// TwinCAT 3 PLC project plc_kfe_gatt
// ProgramVersion: 3.1.4023.0
// libraries:
//   L2SI Vacuum Library, * (SLAC)
//   LCLS General, * (SLAC)
//   lcls-twincat-motion, * (SLAC)
//   PMPS, * (SLAC - LCLS)
//   Tc2_ControllerToolbox, * (Beckhoff Automation GmbH)
//   Tc2_EtherCAT, * (Beckhoff Automation GmbH)
//   Tc2_MC2, * (Beckhoff Automation GmbH)
//   Tc2_Standard, * (Beckhoff Automation GmbH)
//   Tc2_System, * (Beckhoff Automation GmbH)
//   Tc2_Utilities, * (Beckhoff Automation GmbH)
//   Tc3_Module, * (Beckhoff Automation GmbH)
// project tree:
//   DUTs/ E_HomeState.TcDUT, E_MoveState.TcDUT, ST_VGP.TcDUT
//   GVLs/ GVL_Devices.TcGVL, GVL_GATT.TcGVL, GVL_ILK.TcGVL, GVL_MOT.TcGVL, GVL_Variables.TcGVL, Main.TcGVL
//   / PlcTask.TcTTO
//   POUs/ DIAGNOSTICS.TcPOU, FB_MAA_States.TcPOU, FB_VGP.TcPOU, PRG_1_PlcTask.TcPOU, PRG_GATT.TcPOU, PRG_INJ.TcPOU, PRG_Motion.TcPOU, PRG_Motors_Test.TcPOU, PRG_VGP.TcPOU
// real-time tasks:
//   TASK PlcTask: cycle T#10ms, priority 20, ADS port 350
// motion (NC):
//   TASK NC-Task 1 SAF: cycle T#2ms, priority 4, ADS port 501
//   TASK NC-Task 1 SVB: cycle T#10ms, priority 8, ADS port 511
//   AXIS MA_1_X (id 1)
//     Velo: Maximum=5
//     OtherSettings: AllowMotionCmdToSlave=true
//     encoder EncType=4
//       EncPara: ScaleFactorNumerator=6.1991875e-05, MaxCount=#x0000ffff
//         Inc: RefSoftSyncMask=#x0000ffff
//     drive DrvType=24
//       Analog: VeloReferenz=7.93496, TorqueScale=10, ScaleFactorActTorque=0.1
//       TimeComp: TaskDelayCycles=1
//     controller CtrType=1
//       CtrPara: PriorControlFactor=1
//         Observer: BandWidth=20
//   AXIS MA_1_Y (id 2)
//     Dynamic: AccelerationMaximum=30, DecelerationMaximum=30
//     Velo: Maximum=40
//     OtherSettings: AllowMotionCmdToSlave=true
//     encoder EncType=4
//       EncPara: ScaleFactorNumerator=0.000390625, MaxCount=#x0000ffff
//         Inc: RefSoftSyncMask=#x0000ffff
//     drive DrvType=24
//       Analog: VeloReferenz=50, TorqueScale=10, ScaleFactorActTorque=0.1
//       TimeComp: TaskDelayCycles=1
//     controller CtrType=1
//       CtrPara: PriorControlFactor=1
//         Observer: BandWidth=20
//   AXIS MA_2_X (id 3)
//     Velo: Maximum=5
//     OtherSettings: AllowMotionCmdToSlave=true
//     encoder EncType=4
//       EncPara: ScaleFactorNumerator=6.1991875e-05, MaxCount=#x0000ffff
//         Inc: RefSoftSyncMask=#x0000ffff
//     drive DrvType=24
//       Analog: VeloReferenz=7.93496, TorqueScale=10, ScaleFactorActTorque=0.1
//       TimeComp: TaskDelayCycles=1
//     controller CtrType=1
//       CtrPara: PriorControlFactor=1
//         Observer: BandWidth=20
//   AXIS MA_2_Y (id 4)
//     Dynamic: AccelerationMaximum=30, DecelerationMaximum=30
//     Velo: Maximum=40
//     OtherSettings: AllowMotionCmdToSlave=true
//     encoder EncType=4
//       EncPara: ScaleFactorNumerator=0.000390625, MaxCount=#x0000ffff
//         Inc: RefSoftSyncMask=#x0000ffff
//     drive DrvType=24
//       Analog: VeloReferenz=50, TorqueScale=10, ScaleFactorActTorque=0.1
//       TimeComp: TaskDelayCycles=1
//     controller CtrType=1
//       CtrPara: PriorControlFactor=1
//         Observer: BandWidth=20
//   AXIS MA_3_X (id 5)
//     Velo: Maximum=5
//     OtherSettings: AllowMotionCmdToSlave=true
//     encoder EncType=4
//       EncPara: ScaleFactorNumerator=6.1991875e-05, MaxCount=#x0000ffff
//         Inc: RefSoftSyncMask=#x0000ffff
//     drive DrvType=24
//       Analog: VeloReferenz=7.93496, TorqueScale=10, ScaleFactorActTorque=0.1
//       TimeComp: TaskDelayCycles=1
//     controller CtrType=1
//       CtrPara: PriorControlFactor=1
//         Observer: BandWidth=20
//   AXIS MA_3_Y (id 6)
//     Dynamic: AccelerationMaximum=30, DecelerationMaximum=30
//     Velo: Maximum=40
//     OtherSettings: AllowMotionCmdToSlave=true
//     encoder EncType=4
//       EncPara: ScaleFactorNumerator=0.000390625, MaxCount=#x0000ffff
//         Inc: RefSoftSyncMask=#x0000ffff
//     drive DrvType=24
//       Analog: VeloReferenz=50, TorqueScale=10, ScaleFactorActTorque=0.1
//       TimeComp: TaskDelayCycles=1
//     controller CtrType=1
//       CtrPara: PriorControlFactor=1
//         Observer: BandWidth=20
//   AXIS MA_4_X (id 7)
//     Velo: Maximum=5
//     OtherSettings: AllowMotionCmdToSlave=true
//     encoder EncType=4
//       EncPara: ScaleFactorNumerator=6.1991875e-05, MaxCount=#x0000ffff
//         Inc: RefSoftSyncMask=#x0000ffff
//     drive DrvType=24
//       Analog: VeloReferenz=7.93496, TorqueScale=10, ScaleFactorActTorque=0.1
//       TimeComp: TaskDelayCycles=1
//     controller CtrType=1
//       CtrPara: PriorControlFactor=1
//         Observer: BandWidth=20
//   AXIS MA_4_Y (id 8)
//     Dynamic: AccelerationMaximum=30, DecelerationMaximum=30
//     Velo: Maximum=40
//     OtherSettings: AllowMotionCmdToSlave=true
//     encoder EncType=4
//       EncPara: ScaleFactorNumerator=0.000390625, MaxCount=#x0000ffff
//         Inc: RefSoftSyncMask=#x0000ffff
//     drive DrvType=24
//       Analog: VeloReferenz=50, TorqueScale=10, ScaleFactorActTorque=0.1
//       TimeComp: TaskDelayCycles=1
//     controller CtrType=1
//       CtrPara: PriorControlFactor=1
//         Observer: BandWidth=20
//   AXIS VGP_80 (id 9)
//     Velo: Maximum=1800
//     OtherSettings: AllowMotionCmdToSlave=true
//     encoder EncType=4
//       EncPara: ScaleFactorNumerator=0.0390625, Inverse=true, MaxCount=#x0000ffff
//         Inc: RefSoftSyncMask=#x0000ffff
//     drive DrvType=24
//       Analog: VeloReferenz=2000, TorqueScale=10, ScaleFactorActTorque=0.1
//       TimeComp: TaskDelayCycles=1
//     controller CtrType=1
//       CtrPara: PriorControlFactor=1
//         Observer: BandWidth=20
// I/O:
//   DEVICE =+-CX2020/EtherCAT1, AmsNetId 172.21.92.57.2.1
//     =+-EK1200_00_00 [EK1200-5000 EtherCAT Power supply (2A E-Bus)]
//       =+-ES3064_00_01 [EL3064 4Ch. Ana. Input 0-10V]
//       =+-ES9070_00_02 [EL9070 Shield terminal]
//       =+-ES1008_00_03 [EL1008 8Ch. Dig. Input 24V, 3ms]
//       =+-ES2008_00_05 [EL2008 8Ch. Dig. Output 24V, 0.5A]
//       =+-EL2794_00_06 [EL2794 4Ch. Dig. Output 24V AC/DC, 2A, short-circuit-proof]
//       =+-ES2202_00_07 [EL2202 2Ch. Dig. Output 24V, 0.5A]
//       =+-EL6692_00_08 [EL6692 EtherCAT Bridge terminal (Primary)]
//       =+-EK1110_00_09 [EK1110 EtherCAT extension]
//     =+-EK1100_01_00 [EK1100 EtherCAT Coupler (2A E-Bus)]
//       =+-ES3064_01_01 [EL3064 4Ch. Ana. Input 0-10V]
//       =+-ES3064_01_02 [EL3064 4Ch. Ana. Input 0-10V]
//       =+-EL2798_01_03 [EL2798 8Ch. Dig. Output 24V AC/DC, 2A, potential-free]
//       =+-ES3064_01_04 [EL3064 4Ch. Ana. Input 0-10V]
//       =+-ES3064_01_05 [EL3064 4Ch. Ana. Input 0-10V]
//       =+-ES3064_01_06 [EL3064 4Ch. Ana. Input 0-10V]
//       =+-ES3064_01_07 [EL3064 4Ch. Ana. Input 0-10V]
//       =+-EL2798_01_08 [EL2798 8Ch. Dig. Output 24V AC/DC, 2A, potential-free]
//       =+-ES3064_01_09 [EL3064 4Ch. Ana. Input 0-10V]
//       =+-ES3064_01_10 [EL3064 4Ch. Ana. Input 0-10V]
//       =+-EL9410_01_11 [EL9410 E-Bus Power Supplier  (Diagnostics)]
//       =+-ES3064_01_12 [EL3064 4Ch. Ana. Input 0-10V]
//       =+-ES3064_01_13 [EL3064 4Ch. Ana. Input 0-10V]
//       =+-EL2798_01_14 [EL2798 8Ch. Dig. Output 24V AC/DC, 2A, potential-free]
//       =+-ES3064_01_15 [EL3064 4Ch. Ana. Input 0-10V]
//       =+-ES3064_01_16 [EL3064 4Ch. Ana. Input 0-10V]
//       =+-ES3064_01_17 [EL3064 4Ch. Ana. Input 0-10V]
//       =+-ES3064_01_18 [EL3064 4Ch. Ana. Input 0-10V]
//       =+-EL2798_01_19 [EL2798 8Ch. Dig. Output 24V AC/DC, 2A, potential-free]
//       =+-ES3064_01_20 [EL3064 4Ch. Ana. Input 0-10V]
//       =+-ES3064_01_21 [EL3064 4Ch. Ana. Input 0-10V]
//       =+-EK1110_01_22 [EK1110 EtherCAT extension]
//     =+-EK1100_02_00 [EK1100 EtherCAT Coupler (2A E-Bus)]
//       =+-ES2004_02_01 [EL2004 4Ch. Dig. Output 24V, 0.5A]
//       =+-ES1004_02_02 [EL1004 4Ch. Dig. Input 24V, 3ms]
//       =+-ES2004_02_03 [EL2004 4Ch. Dig. Output 24V, 0.5A]
//       =+-ES1004_02_04 [EL1004 4Ch. Dig. Input 24V, 3ms]
//       =+-ES7041_02_05 [EL7041 1Ch. Stepper motor output stage (50V, 5A)]
//       =+-ES7041_02_06 [EL7041 1Ch. Stepper motor output stage (50V, 5A)]
//       =+-ES2004_02_07 [EL2004 4Ch. Dig. Output 24V, 0.5A]
//       =+-ES1004_02_08 [EL1004 4Ch. Dig. Input 24V, 3ms]
//       =+-ES7041_02_09 [EL7041 1Ch. Stepper motor output stage (50V, 5A)]
//       =+-ES7041_02_10 [EL7041 1Ch. Stepper motor output stage (50V, 5A)]
//       =+-ES3064_02_11 [EL3064 4Ch. Ana. Input 0-10V]
//       =+-ES9070_02_12 [EL9070 Shield terminal]
//       =+-ES1008_02_13 [EL1008 8Ch. Dig. Input 24V, 3ms]
//       =+-ES2008_02_14 [EL2008 8Ch. Dig. Output 24V, 0.5A]
//       =+-EL2794_02_15 [EL2794 4Ch. Dig. Output 24V AC/DC, 2A, short-circuit-proof]
//       =+-EL9184_02_16 [EL9184 Potential Connection, 8 x 24V, 8 x Ground]
//       =+-ES3054_02_17 [EL3054 4Ch. Ana. Input 4-20mA]
//       =+-ES6021_02_18 [EL6021 Interface (RS422/485)]
//       =+-EL9011_02_19 [EL9011 End Terminal]
//     =+-EK1100_03_00 [EK1100 EtherCAT Coupler (2A E-Bus)]
//       =+-ES1004_03_01 [EL1004 4Ch. Dig. Input 24V, 3ms]
//       =+-ES1004_03_02 [EL1004 4Ch. Dig. Input 24V, 3ms]
//       =+-EL2798_03_03 [EL2798 8Ch. Dig. Output 24V AC/DC, 2A, potential-free]
//       =+-ES3064_03_04 [EL3064 4Ch. Ana. Input 0-10V]
//       =+-ES4004_03_05 [EL4004 4Ch. Ana. Output 0-10V, 12bit]
//       =+-ES3064_03_06 [EL3064 4Ch. Ana. Input 0-10V]
//       =+-EL2798_03_07 [EL2798 8Ch. Dig. Output 24V AC/DC, 2A, potential-free]
//       =+-ES1004_03_08 [EL1004 4Ch. Dig. Input 24V, 3ms]
//       =+-ES1004_03_09 [EL1004 4Ch. Dig. Input 24V, 3ms]
//       =+-EL9410_03_10 [EL9410 E-Bus Power Supplier  (Diagnostics)]
//       =+-ES1004_03_11 [EL1004 4Ch. Dig. Input 24V, 3ms]
//       =+-ES1004_03_12 [EL1004 4Ch. Dig. Input 24V, 3ms]
//       =+-EL2798_03_13 [EL2798 8Ch. Dig. Output 24V AC/DC, 2A, potential-free]
//       =+-ES3064_03_14 [EL3064 4Ch. Ana. Input 0-10V]
//       =+-ES4004_03_15 [EL4004 4Ch. Ana. Output 0-10V, 12bit]
//       =+-ES3064_03_16 [EL3064 4Ch. Ana. Input 0-10V]
//       =+-EL2798_03_17 [EL2798 8Ch. Dig. Output 24V AC/DC, 2A, potential-free]
//       =+-ES1004_03_18 [EL1004 4Ch. Dig. Input 24V, 3ms]
//       =+-ES1004_03_19 [EL1004 4Ch. Dig. Input 24V, 3ms]
//       =+-EL2794_03_20 [EL2794 4Ch. Dig. Output 24V AC/DC, 2A, short-circuit-proof]
//       =+-ES1004_03_21 [EL1004 4Ch. Dig. Input 24V, 3ms]
//       =+-EL9011_03_22 [EL9011 End Terminal]
//     =+-EK1100_04_00 [EK1100 EtherCAT Coupler (2A E-Bus)]
//       =+-ES2004_04_01 [EL2004 4Ch. Dig. Output 24V, 0.5A]
//       =+-ES4004_04_02 [EL4004 4Ch. Ana. Output 0-10V, 12bit]
//       =+-EL9184_04_03 [EL9184 Potential Connection, 8 x 24V, 8 x Ground]
//       =+-EL7041_04_04 [EL7041 1Ch. Stepper motor output stage (50V, 5A)]
//       =+-EL5101_04_05 [EL5101 1Ch. Inc. Encoder 5V]
//       =+-ES1084_04_06 [EL1084 4Ch. Dig. Input 24V, 3ms, negative]
//       =+-EL7041_04_07 [EL7041 1Ch. Stepper motor output stage (50V, 5A)]
//       =+-EL7041_04_08 [EL7041 1Ch. Stepper motor output stage (50V, 5A)]
//       =+-ES2004_04_09 [EL2004 4Ch. Dig. Output 24V, 0.5A]
//       =+-EL7041_04_10 [EL7041 1Ch. Stepper motor output stage (50V, 5A)]
//       =+-EL7041_04_11 [EL7041 1Ch. Stepper motor output stage (50V, 5A)]
//       =+-ES3054_04_12 [EL3054 4Ch. Ana. Input 4-20mA]
//       =+-ES1084_04_13 [EL1084 4Ch. Dig. Input 24V, 3ms, negative]
//       =+-ES6021_04_14 [EL6021 Interface (RS422/485)]
//       =+-EL9184_04_15 [EL9184 Potential Connection, 8 x 24V, 8 x Ground]
//       =+-ES9070_04_16 [EL9070 Shield terminal]
//       =+-EL3174_04_17 [EL3174-0002 4Ch. Ana. Input +/-10V, +/-20mA 16 Bit, Isolated Channels]
//       =+-EL9011_04_18 [EL9011 End Terminal]
//     =+-EK1100_05_00 [EK1100 EtherCAT Coupler (2A E-Bus)]
//       =+-ES1004_05_01 [EL1004 4Ch. Dig. Input 24V, 3ms]
//       =+-ES2004_05_02 [EL2004 4Ch. Dig. Output 24V, 0.5A]
//       =+-ES1004_05_03 [EL1004 4Ch. Dig. Input 24V, 3ms]
//       =+-ES2004_05_04 [EL2004 4Ch. Dig. Output 24V, 0.5A]
//       =+-ES2004_05_05 [EL2004 4Ch. Dig. Output 24V, 0.5A]
//       =+-ES1004_05_06 [EL1004 4Ch. Dig. Input 24V, 3ms]
//       =+-ES2004_05_07 [EL2004 4Ch. Dig. Output 24V, 0.5A]
//       =+-ES1004_05_08 [EL1004 4Ch. Dig. Input 24V, 3ms]
//       =+-ES1004_05_09 [EL1004 4Ch. Dig. Input 24V, 3ms]
//       =+-EL2798_05_10 [EL2798 8Ch. Dig. Output 24V AC/DC, 2A, potential-free]
//       =+-ES1004_05_11 [EL1004 4Ch. Dig. Input 24V, 3ms]
//       =+-EL1084_05_12 [EL1084 4Ch. Dig. Input 24V, 3ms, negative]
//       =+-EL1084_05_13 [EL1084 4Ch. Dig. Input 24V, 3ms, negative]
//       =+-EL9184_05_14 [EL9184 Potential Connection, 8 x 24V, 8 x Ground]
//       =+-ES9070_05_15 [EL9070 Shield terminal]
//       =+-EL3174_05_16 [EL3174-0002 4Ch. Ana. Input +/-10V, +/-20mA 16 Bit, Isolated Channels]
//       =+-EL9011_05_17 [EL9011 End Terminal]
//     =+-EK1100_06_00 [EK1100 EtherCAT Coupler (2A E-Bus)]
//       =+-ES1004_06_01 [EL1004 4Ch. Dig. Input 24V, 3ms]
//       =+-ES1004_06_02 [EL1004 4Ch. Dig. Input 24V, 3ms]
//       =+-EL2798_06_03 [EL2798 8Ch. Dig. Output 24V AC/DC, 2A, potential-free]
//       =+-ES3064_06_04 [EL3064 4Ch. Ana. Input 0-10V]
//       =+-ES4004_06_05 [EL4004 4Ch. Ana. Output 0-10V, 12bit]
//       =+-ES3064_06_06 [EL3064 4Ch. Ana. Input 0-10V]
//       =+-EL2798_06_07 [EL2798 8Ch. Dig. Output 24V AC/DC, 2A, potential-free]
//       =+-ES1004_06_08 [EL1004 4Ch. Dig. Input 24V, 3ms]
//       =+-ES1004_06_09 [EL1004 4Ch. Dig. Input 24V, 3ms]
//       =+-EL9410_06_10 [EL9410 E-Bus Power Supplier  (Diagnostics)]
//       =+-ES1004_06_11 [EL1004 4Ch. Dig. Input 24V, 3ms]
//       =+-ES1004_06_12 [EL1004 4Ch. Dig. Input 24V, 3ms]
//       =+-EL2798_06_13 [EL2798 8Ch. Dig. Output 24V AC/DC, 2A, potential-free]
//       =+-ES3064_06_14 [EL3064 4Ch. Ana. Input 0-10V]
//       =+-ES4004_06_15 [EL4004 4Ch. Ana. Output 0-10V, 12bit]
//       =+-ES3064_06_16 [EL3064 4Ch. Ana. Input 0-10V]
//       =+-EL2798_06_17 [EL2798 8Ch. Dig. Output 24V AC/DC, 2A, potential-free]
//       =+-ES1004_06_18 [EL1004 4Ch. Dig. Input 24V, 3ms]
//       =+-ES1004_06_19 [EL1004 4Ch. Dig. Input 24V, 3ms]
//       =+-ES1088_06_20 [EL1088 8Ch. Dig. Input 24V, 3ms, negative]
//       =+-ES9187_06_21 [EL9187 Potential Connection, 8 x Ground]
//       =+-EL2794_06_22 [EL2794 4Ch. Dig. Output 24V AC/DC, 2A, short-circuit-proof]
//       =+-ES1088_06_23 [EL1088 8Ch. Dig. Input 24V, 3ms, negative]
//       =+-ES9187_06_24 [EL9187 Potential Connection, 8 x Ground]
//       =+-EL2212_06_25 [EL2212 2Ch. dig. output with overexcitation (24V DC, 2.5A, 10A Peak)]
//       =+-EL2212_06_26 [EL2212 2Ch. dig. output with overexcitation (24V DC, 2.5A, 10A Peak)]
//       =+-EL9011_06_25 [EL9011 End Terminal]
// variable links:
//   NC-Task 1 SAF/Axes/MA_1_X <-> =+-CX2020/EtherCAT1/=+-EK1100_02_00/=+-ES7041_02_05
//     Drive/Inputs/In/nState1 @bit 3 <-> STM Status/Status/Error
//     Drive/Inputs/In/nState1 @bit 5 <-> STM Status/Status/Moving negative
//     Drive/Inputs/In/nState1 @bit 4 <-> STM Status/Status/Moving positive
//     Drive/Inputs/In/nState1 @bit 1 <-> STM Status/Status/Ready
//     Drive/Inputs/In/nState1 <-> STM Status/Status/Ready to enable
//     Drive/Inputs/In/nState1 @bit 6 <-> STM Status/Status/Torque reduced
//     Drive/Inputs/In/nState1 @bit 2 <-> STM Status/Status/Warning
//     Drive/Inputs/In/nState2 @bit 3 <-> STM Status/Status/Digital input 1
//     Drive/Inputs/In/nState2 @bit 4 <-> STM Status/Status/Digital input 2
//     Drive/Inputs/In/nState2 @bit 5 <-> STM Status/Status/Sync error
//     Drive/Inputs/In/nState2 @bit 7 <-> STM Status/Status/TxPDO Toggle
//     Drive/Inputs/In/nState4 @bit 1 <-> WcState/InputToggle
//     Drive/Inputs/In/nState4 <-> WcState/WcState
//     Drive/Outputs/Out/nCtrl1 <-> STM Control/Control/Enable
//     Drive/Outputs/Out/nCtrl1 @bit 2 <-> STM Control/Control/Reduce torque
//     Drive/Outputs/Out/nCtrl1 @bit 1 <-> STM Control/Control/Reset
//     Drive/Outputs/Out/nDataOut2[0] <-> STM Velocity/Velocity
//     Enc/Inputs/In/nDataIn1[0] <-> ENC Status compact/Counter value
//     Enc/Inputs/In/nDataIn2[0] <-> ENC Status compact/Latch value
//     Enc/Inputs/In/nState1 @bit 4 <-> ENC Status compact/Status/Counter overflow
//     Enc/Inputs/In/nState1 @bit 3 <-> ENC Status compact/Status/Counter underflow
//     Enc/Inputs/In/nState1 @bit 7 <-> ENC Status compact/Status/Extrapolation stall
//     Enc/Inputs/In/nState1 <-> ENC Status compact/Status/Latch C valid
//     Enc/Inputs/In/nState1 @bit 1 <-> ENC Status compact/Status/Latch extern valid
//     Enc/Inputs/In/nState1 @bit 2 <-> ENC Status compact/Status/Set counter done
//     Enc/Inputs/In/nState2 @bit 4 <-> ENC Status compact/Status/Status of extern latch
//     Enc/Inputs/In/nState2 <-> ENC Status compact/Status/Status of input A
//     Enc/Inputs/In/nState2 @bit 1 <-> ENC Status compact/Status/Status of input B
//     Enc/Inputs/In/nState2 @bit 2 <-> ENC Status compact/Status/Status of input C
//     Enc/Inputs/In/nState2 @bit 5 <-> ENC Status compact/Status/Sync error
//     Enc/Inputs/In/nState2 @bit 7 <-> ENC Status compact/Status/TxPDO Toggle
//     Enc/Inputs/In/nState4 @bit 1 <-> WcState/InputToggle
//     Enc/Inputs/In/nState4 <-> WcState/WcState
//     Enc/Outputs/Out/nCtrl1 <-> ENC Control compact/Control/Enable latch C
//     Enc/Outputs/Out/nCtrl1 @bit 3 <-> ENC Control compact/Control/Enable latch extern on negative edge
//     Enc/Outputs/Out/nCtrl1 @bit 1 <-> ENC Control compact/Control/Enable latch extern on positive edge
//     Enc/Outputs/Out/nCtrl1 @bit 2 <-> ENC Control compact/Control/Set counter
//     Enc/Outputs/Out/nDataOut1[0] <-> ENC Control compact/Set counter value
//   NC-Task 1 SAF/Axes/MA_1_Y <-> =+-CX2020/EtherCAT1/=+-EK1100_02_00/=+-ES7041_02_06
//     Drive/Inputs/In/nState1 @bit 3 <-> STM Status/Status/Error
//     Drive/Inputs/In/nState1 @bit 5 <-> STM Status/Status/Moving negative
//     Drive/Inputs/In/nState1 @bit 4 <-> STM Status/Status/Moving positive
//     Drive/Inputs/In/nState1 @bit 1 <-> STM Status/Status/Ready
//     Drive/Inputs/In/nState1 <-> STM Status/Status/Ready to enable
//     Drive/Inputs/In/nState1 @bit 6 <-> STM Status/Status/Torque reduced
//     Drive/Inputs/In/nState1 @bit 2 <-> STM Status/Status/Warning
//     Drive/Inputs/In/nState2 @bit 3 <-> STM Status/Status/Digital input 1
//     Drive/Inputs/In/nState2 @bit 4 <-> STM Status/Status/Digital input 2
//     Drive/Inputs/In/nState2 @bit 5 <-> STM Status/Status/Sync error
//     Drive/Inputs/In/nState2 @bit 7 <-> STM Status/Status/TxPDO Toggle
//     Drive/Inputs/In/nState4 @bit 1 <-> WcState/InputToggle
//     Drive/Inputs/In/nState4 <-> WcState/WcState
//     Drive/Outputs/Out/nCtrl1 <-> STM Control/Control/Enable
//     Drive/Outputs/Out/nCtrl1 @bit 2 <-> STM Control/Control/Reduce torque
//     Drive/Outputs/Out/nCtrl1 @bit 1 <-> STM Control/Control/Reset
//     Drive/Outputs/Out/nDataOut2[0] <-> STM Velocity/Velocity
//     Enc/Inputs/In/nDataIn1[0] <-> ENC Status compact/Counter value
//     Enc/Inputs/In/nDataIn2[0] <-> ENC Status compact/Latch value
//     Enc/Inputs/In/nState1 @bit 4 <-> ENC Status compact/Status/Counter overflow
//     Enc/Inputs/In/nState1 @bit 3 <-> ENC Status compact/Status/Counter underflow
//     Enc/Inputs/In/nState1 @bit 7 <-> ENC Status compact/Status/Extrapolation stall
//     Enc/Inputs/In/nState1 <-> ENC Status compact/Status/Latch C valid
//     Enc/Inputs/In/nState1 @bit 1 <-> ENC Status compact/Status/Latch extern valid
//     Enc/Inputs/In/nState1 @bit 2 <-> ENC Status compact/Status/Set counter done
//     Enc/Inputs/In/nState2 @bit 4 <-> ENC Status compact/Status/Status of extern latch
//     Enc/Inputs/In/nState2 <-> ENC Status compact/Status/Status of input A
//     Enc/Inputs/In/nState2 @bit 1 <-> ENC Status compact/Status/Status of input B
//     Enc/Inputs/In/nState2 @bit 2 <-> ENC Status compact/Status/Status of input C
//     Enc/Inputs/In/nState2 @bit 5 <-> ENC Status compact/Status/Sync error
//     Enc/Inputs/In/nState2 @bit 7 <-> ENC Status compact/Status/TxPDO Toggle
//     Enc/Inputs/In/nState4 @bit 1 <-> WcState/InputToggle
//     Enc/Inputs/In/nState4 <-> WcState/WcState
//     Enc/Outputs/Out/nCtrl1 <-> ENC Control compact/Control/Enable latch C
//     Enc/Outputs/Out/nCtrl1 @bit 3 <-> ENC Control compact/Control/Enable latch extern on negative edge
//     Enc/Outputs/Out/nCtrl1 @bit 1 <-> ENC Control compact/Control/Enable latch extern on positive edge
//     Enc/Outputs/Out/nCtrl1 @bit 2 <-> ENC Control compact/Control/Set counter
//     Enc/Outputs/Out/nDataOut1[0] <-> ENC Control compact/Set counter value
//   NC-Task 1 SAF/Axes/MA_2_X <-> =+-CX2020/EtherCAT1/=+-EK1100_02_00/=+-ES7041_02_09
//     Drive/Inputs/In/nState1 @bit 3 <-> STM Status/Status/Error
//     Drive/Inputs/In/nState1 @bit 5 <-> STM Status/Status/Moving negative
//     Drive/Inputs/In/nState1 @bit 4 <-> STM Status/Status/Moving positive
//     Drive/Inputs/In/nState1 @bit 1 <-> STM Status/Status/Ready
//     Drive/Inputs/In/nState1 <-> STM Status/Status/Ready to enable
//     Drive/Inputs/In/nState1 @bit 6 <-> STM Status/Status/Torque reduced
//     Drive/Inputs/In/nState1 @bit 2 <-> STM Status/Status/Warning
//     Drive/Inputs/In/nState2 @bit 3 <-> STM Status/Status/Digital input 1
//     Drive/Inputs/In/nState2 @bit 4 <-> STM Status/Status/Digital input 2
//     Drive/Inputs/In/nState2 @bit 5 <-> STM Status/Status/Sync error
//     Drive/Inputs/In/nState2 @bit 7 <-> STM Status/Status/TxPDO Toggle
//     Drive/Inputs/In/nState4 @bit 1 <-> WcState/InputToggle
//     Drive/Inputs/In/nState4 <-> WcState/WcState
//     Drive/Outputs/Out/nCtrl1 <-> STM Control/Control/Enable
//     Drive/Outputs/Out/nCtrl1 @bit 2 <-> STM Control/Control/Reduce torque
//     Drive/Outputs/Out/nCtrl1 @bit 1 <-> STM Control/Control/Reset
//     Drive/Outputs/Out/nDataOut2[0] <-> STM Velocity/Velocity
//     Enc/Inputs/In/nDataIn1[0] <-> ENC Status compact/Counter value
//     Enc/Inputs/In/nDataIn2[0] <-> ENC Status compact/Latch value
//     Enc/Inputs/In/nState1 @bit 4 <-> ENC Status compact/Status/Counter overflow
//     Enc/Inputs/In/nState1 @bit 3 <-> ENC Status compact/Status/Counter underflow
//     Enc/Inputs/In/nState1 @bit 7 <-> ENC Status compact/Status/Extrapolation stall
//     Enc/Inputs/In/nState1 <-> ENC Status compact/Status/Latch C valid
//     Enc/Inputs/In/nState1 @bit 1 <-> ENC Status compact/Status/Latch extern valid
//     Enc/Inputs/In/nState1 @bit 2 <-> ENC Status compact/Status/Set counter done
//     Enc/Inputs/In/nState2 @bit 4 <-> ENC Status compact/Status/Status of extern latch
//     Enc/Inputs/In/nState2 <-> ENC Status compact/Status/Status of input A
//     Enc/Inputs/In/nState2 @bit 1 <-> ENC Status compact/Status/Status of input B
//     Enc/Inputs/In/nState2 @bit 2 <-> ENC Status compact/Status/Status of input C
//     Enc/Inputs/In/nState2 @bit 5 <-> ENC Status compact/Status/Sync error
//     Enc/Inputs/In/nState2 @bit 7 <-> ENC Status compact/Status/TxPDO Toggle
//     Enc/Inputs/In/nState4 @bit 1 <-> WcState/InputToggle
//     Enc/Inputs/In/nState4 <-> WcState/WcState
//     Enc/Outputs/Out/nCtrl1 <-> ENC Control compact/Control/Enable latch C
//     Enc/Outputs/Out/nCtrl1 @bit 3 <-> ENC Control compact/Control/Enable latch extern on negative edge
//     Enc/Outputs/Out/nCtrl1 @bit 1 <-> ENC Control compact/Control/Enable latch extern on positive edge
//     Enc/Outputs/Out/nCtrl1 @bit 2 <-> ENC Control compact/Control/Set counter
//     Enc/Outputs/Out/nDataOut1[0] <-> ENC Control compact/Set counter value
//   NC-Task 1 SAF/Axes/MA_2_Y <-> =+-CX2020/EtherCAT1/=+-EK1100_02_00/=+-ES7041_02_10
//     Drive/Inputs/In/nState1 @bit 3 <-> STM Status/Status/Error
//     Drive/Inputs/In/nState1 @bit 5 <-> STM Status/Status/Moving negative
//     Drive/Inputs/In/nState1 @bit 4 <-> STM Status/Status/Moving positive
//     Drive/Inputs/In/nState1 @bit 1 <-> STM Status/Status/Ready
//     Drive/Inputs/In/nState1 <-> STM Status/Status/Ready to enable
//     Drive/Inputs/In/nState1 @bit 6 <-> STM Status/Status/Torque reduced
//     Drive/Inputs/In/nState1 @bit 2 <-> STM Status/Status/Warning
//     Drive/Inputs/In/nState2 @bit 3 <-> STM Status/Status/Digital input 1
//     Drive/Inputs/In/nState2 @bit 4 <-> STM Status/Status/Digital input 2
//     Drive/Inputs/In/nState2 @bit 5 <-> STM Status/Status/Sync error
//     Drive/Inputs/In/nState2 @bit 7 <-> STM Status/Status/TxPDO Toggle
//     Drive/Inputs/In/nState4 @bit 1 <-> WcState/InputToggle
//     Drive/Inputs/In/nState4 <-> WcState/WcState
//     Drive/Outputs/Out/nCtrl1 <-> STM Control/Control/Enable
//     Drive/Outputs/Out/nCtrl1 @bit 2 <-> STM Control/Control/Reduce torque
//     Drive/Outputs/Out/nCtrl1 @bit 1 <-> STM Control/Control/Reset
//     Drive/Outputs/Out/nDataOut2[0] <-> STM Velocity/Velocity
//     Enc/Inputs/In/nDataIn1[0] <-> ENC Status compact/Counter value
//     Enc/Inputs/In/nDataIn2[0] <-> ENC Status compact/Latch value
//     Enc/Inputs/In/nState1 @bit 4 <-> ENC Status compact/Status/Counter overflow
//     Enc/Inputs/In/nState1 @bit 3 <-> ENC Status compact/Status/Counter underflow
//     Enc/Inputs/In/nState1 @bit 7 <-> ENC Status compact/Status/Extrapolation stall
//     Enc/Inputs/In/nState1 <-> ENC Status compact/Status/Latch C valid
//     Enc/Inputs/In/nState1 @bit 1 <-> ENC Status compact/Status/Latch extern valid
//     Enc/Inputs/In/nState1 @bit 2 <-> ENC Status compact/Status/Set counter done
//     Enc/Inputs/In/nState2 @bit 4 <-> ENC Status compact/Status/Status of extern latch
//     Enc/Inputs/In/nState2 <-> ENC Status compact/Status/Status of input A
//     Enc/Inputs/In/nState2 @bit 1 <-> ENC Status compact/Status/Status of input B
//     Enc/Inputs/In/nState2 @bit 2 <-> ENC Status compact/Status/Status of input C
//     Enc/Inputs/In/nState2 @bit 5 <-> ENC Status compact/Status/Sync error
//     Enc/Inputs/In/nState2 @bit 7 <-> ENC Status compact/Status/TxPDO Toggle
//     Enc/Inputs/In/nState4 @bit 1 <-> WcState/InputToggle
//     Enc/Inputs/In/nState4 <-> WcState/WcState
//     Enc/Outputs/Out/nCtrl1 <-> ENC Control compact/Control/Enable latch C
//     Enc/Outputs/Out/nCtrl1 @bit 3 <-> ENC Control compact/Control/Enable latch extern on negative edge
//     Enc/Outputs/Out/nCtrl1 @bit 1 <-> ENC Control compact/Control/Enable latch extern on positive edge
//     Enc/Outputs/Out/nCtrl1 @bit 2 <-> ENC Control compact/Control/Set counter
//     Enc/Outputs/Out/nDataOut1[0] <-> ENC Control compact/Set counter value
//   NC-Task 1 SAF/Axes/MA_3_X <-> =+-CX2020/EtherCAT1/=+-EK1100_04_00/=+-EL7041_04_07
//     Drive/Inputs/In/nState1 @bit 3 <-> STM Status/Status/Error
//     Drive/Inputs/In/nState1 @bit 5 <-> STM Status/Status/Moving negative
//     Drive/Inputs/In/nState1 @bit 4 <-> STM Status/Status/Moving positive
//     Drive/Inputs/In/nState1 @bit 1 <-> STM Status/Status/Ready
//     Drive/Inputs/In/nState1 <-> STM Status/Status/Ready to enable
//     Drive/Inputs/In/nState1 @bit 6 <-> STM Status/Status/Torque reduced
//     Drive/Inputs/In/nState1 @bit 2 <-> STM Status/Status/Warning
//     Drive/Inputs/In/nState2 @bit 3 <-> STM Status/Status/Digital input 1
//     Drive/Inputs/In/nState2 @bit 4 <-> STM Status/Status/Digital input 2
//     Drive/Inputs/In/nState2 @bit 5 <-> STM Status/Status/Sync error
//     Drive/Inputs/In/nState2 @bit 7 <-> STM Status/Status/TxPDO Toggle
//     Drive/Inputs/In/nState4 @bit 1 <-> WcState/InputToggle
//     Drive/Inputs/In/nState4 <-> WcState/WcState
//     Drive/Outputs/Out/nCtrl1 <-> STM Control/Control/Enable
//     Drive/Outputs/Out/nCtrl1 @bit 2 <-> STM Control/Control/Reduce torque
//     Drive/Outputs/Out/nCtrl1 @bit 1 <-> STM Control/Control/Reset
//     Drive/Outputs/Out/nDataOut2[0] <-> STM Velocity/Velocity
//     Enc/Inputs/In/nDataIn1[0] <-> ENC Status compact/Counter value
//     Enc/Inputs/In/nDataIn2[0] <-> ENC Status compact/Latch value
//     Enc/Inputs/In/nState1 @bit 4 <-> ENC Status compact/Status/Counter overflow
//     Enc/Inputs/In/nState1 @bit 3 <-> ENC Status compact/Status/Counter underflow
//     Enc/Inputs/In/nState1 @bit 7 <-> ENC Status compact/Status/Extrapolation stall
//     Enc/Inputs/In/nState1 <-> ENC Status compact/Status/Latch C valid
//     Enc/Inputs/In/nState1 @bit 1 <-> ENC Status compact/Status/Latch extern valid
//     Enc/Inputs/In/nState1 @bit 2 <-> ENC Status compact/Status/Set counter done
//     Enc/Inputs/In/nState2 @bit 4 <-> ENC Status compact/Status/Status of extern latch
//     Enc/Inputs/In/nState2 <-> ENC Status compact/Status/Status of input A
//     Enc/Inputs/In/nState2 @bit 1 <-> ENC Status compact/Status/Status of input B
//     Enc/Inputs/In/nState2 @bit 2 <-> ENC Status compact/Status/Status of input C
//     Enc/Inputs/In/nState2 @bit 5 <-> ENC Status compact/Status/Sync error
//     Enc/Inputs/In/nState2 @bit 7 <-> ENC Status compact/Status/TxPDO Toggle
//     Enc/Inputs/In/nState4 @bit 1 <-> WcState/InputToggle
//     Enc/Inputs/In/nState4 <-> WcState/WcState
//     Enc/Outputs/Out/nCtrl1 <-> ENC Control compact/Control/Enable latch C
//     Enc/Outputs/Out/nCtrl1 @bit 3 <-> ENC Control compact/Control/Enable latch extern on negative edge
//     Enc/Outputs/Out/nCtrl1 @bit 1 <-> ENC Control compact/Control/Enable latch extern on positive edge
//     Enc/Outputs/Out/nCtrl1 @bit 2 <-> ENC Control compact/Control/Set counter
//     Enc/Outputs/Out/nDataOut1[0] <-> ENC Control compact/Set counter value
//   NC-Task 1 SAF/Axes/MA_3_Y <-> =+-CX2020/EtherCAT1/=+-EK1100_04_00/=+-EL7041_04_08
//     Drive/Inputs/In/nState1 @bit 3 <-> STM Status/Status/Error
//     Drive/Inputs/In/nState1 @bit 5 <-> STM Status/Status/Moving negative
//     Drive/Inputs/In/nState1 @bit 4 <-> STM Status/Status/Moving positive
//     Drive/Inputs/In/nState1 @bit 1 <-> STM Status/Status/Ready
//     Drive/Inputs/In/nState1 <-> STM Status/Status/Ready to enable
//     Drive/Inputs/In/nState1 @bit 6 <-> STM Status/Status/Torque reduced
//     Drive/Inputs/In/nState1 @bit 2 <-> STM Status/Status/Warning
//     Drive/Inputs/In/nState2 @bit 3 <-> STM Status/Status/Digital input 1
//     Drive/Inputs/In/nState2 @bit 4 <-> STM Status/Status/Digital input 2
//     Drive/Inputs/In/nState2 @bit 5 <-> STM Status/Status/Sync error
//     Drive/Inputs/In/nState2 @bit 7 <-> STM Status/Status/TxPDO Toggle
//     Drive/Inputs/In/nState4 @bit 1 <-> WcState/InputToggle
//     Drive/Inputs/In/nState4 <-> WcState/WcState
//     Drive/Outputs/Out/nCtrl1 <-> STM Control/Control/Enable
//     Drive/Outputs/Out/nCtrl1 @bit 2 <-> STM Control/Control/Reduce torque
//     Drive/Outputs/Out/nCtrl1 @bit 1 <-> STM Control/Control/Reset
//     Drive/Outputs/Out/nDataOut2[0] <-> STM Velocity/Velocity
//     Enc/Inputs/In/nDataIn1[0] <-> ENC Status compact/Counter value
//     Enc/Inputs/In/nDataIn2[0] <-> ENC Status compact/Latch value
//     Enc/Inputs/In/nState1 @bit 4 <-> ENC Status compact/Status/Counter overflow
//     Enc/Inputs/In/nState1 @bit 3 <-> ENC Status compact/Status/Counter underflow
//     Enc/Inputs/In/nState1 @bit 7 <-> ENC Status compact/Status/Extrapolation stall
//     Enc/Inputs/In/nState1 <-> ENC Status compact/Status/Latch C valid
//     Enc/Inputs/In/nState1 @bit 1 <-> ENC Status compact/Status/Latch extern valid
//     Enc/Inputs/In/nState1 @bit 2 <-> ENC Status compact/Status/Set counter done
//     Enc/Inputs/In/nState2 @bit 4 <-> ENC Status compact/Status/Status of extern latch
//     Enc/Inputs/In/nState2 <-> ENC Status compact/Status/Status of input A
//     Enc/Inputs/In/nState2 @bit 1 <-> ENC Status compact/Status/Status of input B
//     Enc/Inputs/In/nState2 @bit 2 <-> ENC Status compact/Status/Status of input C
//     Enc/Inputs/In/nState2 @bit 5 <-> ENC Status compact/Status/Sync error
//     Enc/Inputs/In/nState2 @bit 7 <-> ENC Status compact/Status/TxPDO Toggle
//     Enc/Inputs/In/nState4 @bit 1 <-> WcState/InputToggle
//     Enc/Inputs/In/nState4 <-> WcState/WcState
//     Enc/Outputs/Out/nCtrl1 <-> ENC Control compact/Control/Enable latch C
//     Enc/Outputs/Out/nCtrl1 @bit 3 <-> ENC Control compact/Control/Enable latch extern on negative edge
//     Enc/Outputs/Out/nCtrl1 @bit 1 <-> ENC Control compact/Control/Enable latch extern on positive edge
//     Enc/Outputs/Out/nCtrl1 @bit 2 <-> ENC Control compact/Control/Set counter
//     Enc/Outputs/Out/nDataOut1[0] <-> ENC Control compact/Set counter value
//   NC-Task 1 SAF/Axes/MA_4_X <-> =+-CX2020/EtherCAT1/=+-EK1100_04_00/=+-EL7041_04_10
//     Drive/Inputs/In/nState1 @bit 3 <-> STM Status/Status/Error
//     Drive/Inputs/In/nState1 @bit 5 <-> STM Status/Status/Moving negative
//     Drive/Inputs/In/nState1 @bit 4 <-> STM Status/Status/Moving positive
//     Drive/Inputs/In/nState1 @bit 1 <-> STM Status/Status/Ready
//     Drive/Inputs/In/nState1 <-> STM Status/Status/Ready to enable
//     Drive/Inputs/In/nState1 @bit 6 <-> STM Status/Status/Torque reduced
//     Drive/Inputs/In/nState1 @bit 2 <-> STM Status/Status/Warning
//     Drive/Inputs/In/nState2 @bit 3 <-> STM Status/Status/Digital input 1
//     Drive/Inputs/In/nState2 @bit 4 <-> STM Status/Status/Digital input 2
//     Drive/Inputs/In/nState2 @bit 5 <-> STM Status/Status/Sync error
//     Drive/Inputs/In/nState2 @bit 7 <-> STM Status/Status/TxPDO Toggle
//     Drive/Inputs/In/nState4 @bit 1 <-> WcState/InputToggle
//     Drive/Inputs/In/nState4 <-> WcState/WcState
//     Drive/Outputs/Out/nCtrl1 <-> STM Control/Control/Enable
//     Drive/Outputs/Out/nCtrl1 @bit 2 <-> STM Control/Control/Reduce torque
//     Drive/Outputs/Out/nCtrl1 @bit 1 <-> STM Control/Control/Reset
//     Drive/Outputs/Out/nDataOut2[0] <-> STM Velocity/Velocity
//     Enc/Inputs/In/nDataIn1[0] <-> ENC Status compact/Counter value
//     Enc/Inputs/In/nDataIn2[0] <-> ENC Status compact/Latch value
//     Enc/Inputs/In/nState1 @bit 4 <-> ENC Status compact/Status/Counter overflow
//     Enc/Inputs/In/nState1 @bit 3 <-> ENC Status compact/Status/Counter underflow
//     Enc/Inputs/In/nState1 @bit 7 <-> ENC Status compact/Status/Extrapolation stall
//     Enc/Inputs/In/nState1 <-> ENC Status compact/Status/Latch C valid
//     Enc/Inputs/In/nState1 @bit 1 <-> ENC Status compact/Status/Latch extern valid
//     Enc/Inputs/In/nState1 @bit 2 <-> ENC Status compact/Status/Set counter done
//     Enc/Inputs/In/nState2 @bit 4 <-> ENC Status compact/Status/Status of extern latch
//     Enc/Inputs/In/nState2 <-> ENC Status compact/Status/Status of input A
//     Enc/Inputs/In/nState2 @bit 1 <-> ENC Status compact/Status/Status of input B
//     Enc/Inputs/In/nState2 @bit 2 <-> ENC Status compact/Status/Status of input C
//     Enc/Inputs/In/nState2 @bit 5 <-> ENC Status compact/Status/Sync error
//     Enc/Inputs/In/nState2 @bit 7 <-> ENC Status compact/Status/TxPDO Toggle
//     Enc/Inputs/In/nState4 @bit 1 <-> WcState/InputToggle
//     Enc/Inputs/In/nState4 <-> WcState/WcState
//     Enc/Outputs/Out/nCtrl1 <-> ENC Control compact/Control/Enable latch C
//     Enc/Outputs/Out/nCtrl1 @bit 3 <-> ENC Control compact/Control/Enable latch extern on negative edge
//     Enc/Outputs/Out/nCtrl1 @bit 1 <-> ENC Control compact/Control/Enable latch extern on positive edge
//     Enc/Outputs/Out/nCtrl1 @bit 2 <-> ENC Control compact/Control/Set counter
//     Enc/Outputs/Out/nDataOut1[0] <-> ENC Control compact/Set counter value
//   NC-Task 1 SAF/Axes/MA_4_Y <-> =+-CX2020/EtherCAT1/=+-EK1100_04_00/=+-EL7041_04_11
//     Drive/Inputs/In/nState1 @bit 3 <-> STM Status/Status/Error
//     Drive/Inputs/In/nState1 @bit 5 <-> STM Status/Status/Moving negative
//     Drive/Inputs/In/nState1 @bit 4 <-> STM Status/Status/Moving positive
//     Drive/Inputs/In/nState1 @bit 1 <-> STM Status/Status/Ready
//     Drive/Inputs/In/nState1 <-> STM Status/Status/Ready to enable
//     Drive/Inputs/In/nState1 @bit 6 <-> STM Status/Status/Torque reduced
//     Drive/Inputs/In/nState1 @bit 2 <-> STM Status/Status/Warning
//     Drive/Inputs/In/nState2 @bit 3 <-> STM Status/Status/Digital input 1
//     Drive/Inputs/In/nState2 @bit 4 <-> STM Status/Status/Digital input 2
//     Drive/Inputs/In/nState2 @bit 5 <-> STM Status/Status/Sync error
//     Drive/Inputs/In/nState2 @bit 7 <-> STM Status/Status/TxPDO Toggle
//     Drive/Inputs/In/nState4 @bit 1 <-> WcState/InputToggle
//     Drive/Inputs/In/nState4 <-> WcState/WcState
//     Drive/Outputs/Out/nCtrl1 <-> STM Control/Control/Enable
//     Drive/Outputs/Out/nCtrl1 @bit 2 <-> STM Control/Control/Reduce torque
//     Drive/Outputs/Out/nCtrl1 @bit 1 <-> STM Control/Control/Reset
//     Drive/Outputs/Out/nDataOut2[0] <-> STM Velocity/Velocity
//     Enc/Inputs/In/nDataIn1[0] <-> ENC Status compact/Counter value
//     Enc/Inputs/In/nDataIn2[0] <-> ENC Status compact/Latch value
//     Enc/Inputs/In/nState1 @bit 4 <-> ENC Status compact/Status/Counter overflow
//     Enc/Inputs/In/nState1 @bit 3 <-> ENC Status compact/Status/Counter underflow
//     Enc/Inputs/In/nState1 @bit 7 <-> ENC Status compact/Status/Extrapolation stall
//     Enc/Inputs/In/nState1 <-> ENC Status compact/Status/Latch C valid
//     Enc/Inputs/In/nState1 @bit 1 <-> ENC Status compact/Status/Latch extern valid
//     Enc/Inputs/In/nState1 @bit 2 <-> ENC Status compact/Status/Set counter done
//     Enc/Inputs/In/nState2 @bit 4 <-> ENC Status compact/Status/Status of extern latch
//     Enc/Inputs/In/nState2 <-> ENC Status compact/Status/Status of input A
//     Enc/Inputs/In/nState2 @bit 1 <-> ENC Status compact/Status/Status of input B
//     Enc/Inputs/In/nState2 @bit 2 <-> ENC Status compact/Status/Status of input C
//     Enc/Inputs/In/nState2 @bit 5 <-> ENC Status compact/Status/Sync error
//     Enc/Inputs/In/nState2 @bit 7 <-> ENC Status compact/Status/TxPDO Toggle
//     Enc/Inputs/In/nState4 @bit 1 <-> WcState/InputToggle
//     Enc/Inputs/In/nState4 <-> WcState/WcState
//     Enc/Outputs/Out/nCtrl1 <-> ENC Control compact/Control/Enable latch C
//     Enc/Outputs/Out/nCtrl1 @bit 3 <-> ENC Control compact/Control/Enable latch extern on negative edge
//     Enc/Outputs/Out/nCtrl1 @bit 1 <-> ENC Control compact/Control/Enable latch extern on positive edge
//     Enc/Outputs/Out/nCtrl1 @bit 2 <-> ENC Control compact/Control/Set counter
//     Enc/Outputs/Out/nDataOut1[0] <-> ENC Control compact/Set counter value
//   NC-Task 1 SAF/Axes/VGP_80 <-> =+-CX2020/EtherCAT1/=+-EK1100_04_00/=+-EL5101_04_05
//     Enc/Inputs/In/nDataIn1[0] <-> ENC Status compact/Counter value
//     Enc/Inputs/In/nDataIn2[0] <-> ENC Status compact/Latch value
//     Enc/Inputs/In/nState1 @bit 4 <-> ENC Status compact/Status/Counter overflow
//     Enc/Inputs/In/nState1 @bit 3 <-> ENC Status compact/Status/Counter underflow
//     Enc/Inputs/In/nState1 @bit 7 <-> ENC Status compact/Status/Extrapolation stall
//     Enc/Inputs/In/nState1 <-> ENC Status compact/Status/Latch C valid
//     Enc/Inputs/In/nState1 @bit 1 <-> ENC Status compact/Status/Latch extern valid
//     Enc/Inputs/In/nState1 @bit 6 <-> ENC Status compact/Status/Open circuit
//     Enc/Inputs/In/nState1 @bit 2 <-> ENC Status compact/Status/Set counter done
//     Enc/Inputs/In/nState1 @bit 5 <-> ENC Status compact/Status/Status of input status
//     Enc/Inputs/In/nState2 @bit 4 <-> ENC Status compact/Status/Status of extern latch
//     Enc/Inputs/In/nState2 <-> ENC Status compact/Status/Status of input A
//     Enc/Inputs/In/nState2 @bit 1 <-> ENC Status compact/Status/Status of input B
//     Enc/Inputs/In/nState2 @bit 2 <-> ENC Status compact/Status/Status of input C
//     Enc/Inputs/In/nState2 @bit 3 <-> ENC Status compact/Status/Status of input gate
//     Enc/Inputs/In/nState2 @bit 5 <-> ENC Status compact/Status/Sync error
//     Enc/Inputs/In/nState2 @bit 6 <-> ENC Status compact/Status/TxPDO State
//     Enc/Inputs/In/nState2 @bit 7 <-> ENC Status compact/Status/TxPDO Toggle
//     Enc/Inputs/In/nState4 @bit 1 <-> WcState/InputToggle
//     Enc/Inputs/In/nState4 <-> WcState/WcState
//     Enc/Outputs/Out/nCtrl1 <-> ENC Control compact/Control/Enable latch C
//     Enc/Outputs/Out/nCtrl1 @bit 3 <-> ENC Control compact/Control/Enable latch extern on negative edge
//     Enc/Outputs/Out/nCtrl1 @bit 1 <-> ENC Control compact/Control/Enable latch extern on positive edge
//     Enc/Outputs/Out/nCtrl1 @bit 2 <-> ENC Control compact/Control/Set counter
//     Enc/Outputs/Out/nDataOut1[0] <-> ENC Control compact/Set counter value
//   NC-Task 1 SAF/Axes/VGP_80 <-> =+-CX2020/EtherCAT1/=+-EK1100_04_00/=+-EL7041_04_04
//     Drive/Inputs/In/nState1 @bit 3 <-> STM Status/Status/Error
//     Drive/Inputs/In/nState1 @bit 5 <-> STM Status/Status/Moving negative
//     Drive/Inputs/In/nState1 @bit 4 <-> STM Status/Status/Moving positive
//     Drive/Inputs/In/nState1 @bit 1 <-> STM Status/Status/Ready
//     Drive/Inputs/In/nState1 <-> STM Status/Status/Ready to enable
//     Drive/Inputs/In/nState1 @bit 6 <-> STM Status/Status/Torque reduced
//     Drive/Inputs/In/nState1 @bit 2 <-> STM Status/Status/Warning
//     Drive/Inputs/In/nState2 @bit 3 <-> STM Status/Status/Digital input 1
//     Drive/Inputs/In/nState2 @bit 4 <-> STM Status/Status/Digital input 2
//     Drive/Inputs/In/nState2 @bit 5 <-> STM Status/Status/Sync error
//     Drive/Inputs/In/nState2 @bit 7 <-> STM Status/Status/TxPDO Toggle
//     Drive/Inputs/In/nState4 @bit 1 <-> WcState/InputToggle
//     Drive/Inputs/In/nState4 <-> WcState/WcState
//     Drive/Outputs/Out/nCtrl1 <-> STM Control/Control/Enable
//     Drive/Outputs/Out/nCtrl1 @bit 2 <-> STM Control/Control/Reduce torque
//     Drive/Outputs/Out/nCtrl1 @bit 1 <-> STM Control/Control/Reset
//     Drive/Outputs/Out/nDataOut2[0] <-> STM Velocity/Velocity
//   plc_kfe_gatt Instance <-> =+-CX2020/EtherCAT1/=+-EK1100_01_00/=+-EL2798_01_03
//     PlcTask Outputs/GVL_Devices.fb_AT1K0_GAS_GCC_10.q_xHV_DIS <-> Channel 1/fb_AT1K0_GAS_GCC_10.q_xHV_DIS
//     PlcTask Outputs/GVL_Devices.fb_AT1K0_GAS_GCC_20.q_xHV_DIS <-> Channel 2/fb_AT1K0_GAS_GCC_20.q_xHV_DIS
//     PlcTask Outputs/GVL_Devices.fb_AT1K0_GAS_GCC_30.q_xHV_DIS <-> Channel 5/fb_AT1K0_GAS_GCC_30.q_xHV_DIS
//     PlcTask Outputs/GVL_Devices.fb_AT1K0_GAS_GCC_40.q_xHV_DIS <-> Channel 6/fb_AT1K0_GAS_GCC_40.q_xHV_DIS
//   plc_kfe_gatt Instance <-> =+-CX2020/EtherCAT1/=+-EK1100_01_00/=+-EL2798_01_08
//     PlcTask Outputs/GVL_Devices.fb_AT1K0_GAS_GCC_50.q_xHV_DIS <-> Channel 1/fb_AT1K0_GAS_GCC_50.q_xHV_DIS
//     PlcTask Outputs/GVL_Devices.fb_AT1K0_GAS_GCC_60.q_xHV_DIS <-> Channel 2/fb_AT1K0_GAS_GCC_60.q_xHV_DIS
//     PlcTask Outputs/GVL_Devices.fb_AT1K0_GAS_GCC_80.q_xHV_DIS <-> Channel 5/fb_AT1K0_GAS_GCC_80.q_xHV_DIS
//   plc_kfe_gatt Instance <-> =+-CX2020/EtherCAT1/=+-EK1100_01_00/=+-EL2798_01_14
//     PlcTask Outputs/GVL_Devices.fb_AT1K0_GAS_GCC_100.q_xHV_DIS <-> Channel 2/fb_AT1K0_GAS_GCC_100.q_xHV_DIS
//     PlcTask Outputs/GVL_Devices.fb_AT1K0_GAS_GCC_110.q_xHV_DIS <-> Channel 5/fb_AT1K0_GAS_GCC_110.q_xHV_DIS
//     PlcTask Outputs/GVL_Devices.fb_AT1K0_GAS_GCC_120.q_xHV_DIS <-> Channel 6/fb_AT1K0_GAS_GCC_120.q_xHV_DIS
//     PlcTask Outputs/GVL_Devices.fb_AT1K0_GAS_GCC_90.q_xHV_DIS <-> Channel 1/fb_AT1K0_GAS_GCC_90.q_xHV_DIS
//   plc_kfe_gatt Instance <-> =+-CX2020/EtherCAT1/=+-EK1100_01_00/=+-EL2798_01_19
//     PlcTask Outputs/GVL_Devices.fb_AT1K0_GAS_GCC_130.q_xHV_DIS <-> Channel 1/Output
//     PlcTask Outputs/GVL_Devices.fb_AT1K0_GAS_GCC_140.q_xHV_DIS <-> Channel 2/Output
//   plc_kfe_gatt Instance <-> =+-CX2020/EtherCAT1/=+-EK1100_01_00/=+-ES3064_01_01
//     PlcTask Inputs/GVL_Devices.fb_AT1K0_GAS_GCC_10.i_iPRESS_R <-> AI Standard Channel 1/fb_AT1K0_GAS_GCC_10.i_iPRESS_R
//     PlcTask Inputs/GVL_Devices.fb_AT1K0_GAS_GCC_20.i_iPRESS_R <-> AI Standard Channel 3/fb_AT1K0_GAS_GCC_20.i_iPRESS_R
//   plc_kfe_gatt Instance <-> =+-CX2020/EtherCAT1/=+-EK1100_01_00/=+-ES3064_01_02
//     PlcTask Inputs/GVL_Devices.fb_AT1K0_GAS_GPI_10.i_iPRESS_R <-> AI Standard Channel 1/fb_AT1K0_GAS_GPI_10.i_iPRESS_R
//     PlcTask Inputs/GVL_Devices.fb_AT1K0_GAS_GPI_20.i_iPRESS_R <-> AI Standard Channel 2/fb_AT1K0_GAS_GPI_20.i_iPRESS_R
//   plc_kfe_gatt Instance <-> =+-CX2020/EtherCAT1/=+-EK1100_01_00/=+-ES3064_01_04
//     PlcTask Inputs/GVL_Devices.fb_AT1K0_GAS_GCC_30.i_iPRESS_R <-> AI Standard Channel 1/fb_AT1K0_GAS_GCC_30.i_iPRESS_R
//     PlcTask Inputs/GVL_Devices.fb_AT1K0_GAS_GCC_40.i_iPRESS_R <-> AI Standard Channel 3/fb_AT1K0_GAS_GCC_40.i_iPRESS_R
//   plc_kfe_gatt Instance <-> =+-CX2020/EtherCAT1/=+-EK1100_01_00/=+-ES3064_01_05
//     PlcTask Inputs/GVL_Devices.fb_AT1K0_GAS_GPI_30.i_iPRESS_R <-> AI Standard Channel 1/fb_AT1K0_GAS_GPI_30.i_iPRESS_R
//     PlcTask Inputs/GVL_Devices.fb_AT1K0_GAS_GPI_40.i_iPRESS_R <-> AI Standard Channel 2/fb_AT1K0_GAS_GPI_40.i_iPRESS_R
//   plc_kfe_gatt Instance <-> =+-CX2020/EtherCAT1/=+-EK1100_01_00/=+-ES3064_01_06
//     PlcTask Inputs/GVL_Devices.fb_AT1K0_GAS_GCC_50.i_iPRESS_R <-> AI Standard Channel 1/fb_AT1K0_GAS_GCC_50.i_iPRESS_R
//     PlcTask Inputs/GVL_Devices.fb_AT1K0_GAS_GCC_60.i_iPRESS_R <-> AI Standard Channel 3/fb_AT1K0_GAS_GCC_60.i_iPRESS_R
//   plc_kfe_gatt Instance <-> =+-CX2020/EtherCAT1/=+-EK1100_01_00/=+-ES3064_01_07
//     PlcTask Inputs/GVL_Devices.fb_AT1K0_GAS_GPI_50.i_iPRESS_R <-> AI Standard Channel 1/fb_AT1K0_GAS_GPI_50.i_iPRESS_R
//     PlcTask Inputs/GVL_Devices.fb_AT1K0_GAS_GPI_60.i_iPRESS_R <-> AI Standard Channel 2/fb_AT1K0_GAS_GPI_60.i_iPRESS_R
//   plc_kfe_gatt Instance <-> =+-CX2020/EtherCAT1/=+-EK1100_01_00/=+-ES3064_01_09
//     PlcTask Inputs/GVL_Devices.fb_AT1K0_GAS_GCC_80.i_iPRESS_R <-> AI Standard Channel 1/fb_AT1K0_GAS_GCC_80.i_iPRESS_R
//     PlcTask Inputs/GVL_Devices.fb_AT1K0_GAS_GPI_80.i_iPRESS_R <-> AI Standard Channel 3/fb_AT1K0_GAS_GPI_80.i_iPRESS_R
//   plc_kfe_gatt Instance <-> =+-CX2020/EtherCAT1/=+-EK1100_01_00/=+-ES3064_01_10
//     PlcTask Inputs/GVL_Devices.fb_AT1K0_GAS_GPI_11.i_iPRESS_R <-> AI Standard Channel 1/fb_AT1K0_GAS_GPI_11.i_iPRESS_R
//     PlcTask Inputs/GVL_Devices.fb_AT1K0_GAS_GPI_51.i_iPRESS_R <-> AI Standard Channel 2/fb_AT1K0_GAS_GPI_51.i_iPRESS_R
//   plc_kfe_gatt Instance <-> =+-CX2020/EtherCAT1/=+-EK1100_01_00/=+-ES3064_01_12
//     PlcTask Inputs/GVL_Devices.fb_AT1K0_GAS_GCC_100.i_iPRESS_R <-> AI Standard Channel 3/fb_AT1K0_GAS_GCC_100.i_iPRESS_R
//     PlcTask Inputs/GVL_Devices.fb_AT1K0_GAS_GCC_90.i_iPRESS_R <-> AI Standard Channel 1/fb_AT1K0_GAS_GCC_90.i_iPRESS_R
//   plc_kfe_gatt Instance <-> =+-CX2020/EtherCAT1/=+-EK1100_01_00/=+-ES3064_01_13
//     PlcTask Inputs/GVL_Devices.fb_AT1K0_GAS_GPI_100.i_iPRESS_R <-> AI Standard Channel 2/fb_AT1K0_GAS_GPI_100.i_iPRESS_R
//     PlcTask Inputs/GVL_Devices.fb_AT1K0_GAS_GPI_90.i_iPRESS_R <-> AI Standard Channel 1/fb_AT1K0_GAS_GPI_90.i_iPRESS_R
//   plc_kfe_gatt Instance <-> =+-CX2020/EtherCAT1/=+-EK1100_01_00/=+-ES3064_01_15
//     PlcTask Inputs/GVL_Devices.fb_AT1K0_GAS_GCC_110.i_iPRESS_R <-> AI Standard Channel 1/fb_AT1K0_GAS_GCC_110.i_iPRESS_R
//     PlcTask Inputs/GVL_Devices.fb_AT1K0_GAS_GCC_120.i_iPRESS_R <-> AI Standard Channel 3/fb_AT1K0_GAS_GCC_120.i_iPRESS_R
//   plc_kfe_gatt Instance <-> =+-CX2020/EtherCAT1/=+-EK1100_01_00/=+-ES3064_01_16
//     PlcTask Inputs/GVL_Devices.fb_AT1K0_GAS_GPI_110.i_iPRESS_R <-> AI Standard Channel 1/fb_AT1K0_GAS_GPI_110.i_iPRESS_R
//     PlcTask Inputs/GVL_Devices.fb_AT1K0_GAS_GPI_120.i_iPRESS_R <-> AI Standard Channel 2/fb_AT1K0_GAS_GPI_120.i_iPRESS_R
//   plc_kfe_gatt Instance <-> =+-CX2020/EtherCAT1/=+-EK1100_01_00/=+-ES3064_01_17
//     PlcTask Inputs/GVL_Devices.fb_AT1K0_GAS_GCC_130.i_iPRESS_R <-> AI Standard Channel 1/fb_AT1K0_GAS_GCC_130.i_iPRESS_R
//     PlcTask Inputs/GVL_Devices.fb_AT1K0_GAS_GCC_140.i_iPRESS_R <-> AI Standard Channel 3/fb_AT1K0_GAS_GCC_140.i_iPRESS_R
//   plc_kfe_gatt Instance <-> =+-CX2020/EtherCAT1/=+-EK1100_01_00/=+-ES3064_01_18
//     PlcTask Inputs/GVL_Devices.fb_AT1K0_GAS_GPI_130.i_iPRESS_R <-> AI Standard Channel 1/fb_AT1K0_GAS_GPI_130.i_iPRESS_R
//     PlcTask Inputs/GVL_Devices.fb_AT1K0_GAS_GPI_140.i_iPRESS_R <-> AI Standard Channel 2/fb_AT1K0_GAS_GPI_140.i_iPRESS_R
//   plc_kfe_gatt Instance <-> =+-CX2020/EtherCAT1/=+-EK1100_02_00/=+-ES1004_02_02
//     PlcTask Inputs/GVL_Devices.fb_AT1K0_GAS_VRC_10.i_xClsLS <-> Channel 2/fb_AT1K0_GAS_VRC_10.i_xClsLS
//     PlcTask Inputs/GVL_Devices.fb_AT1K0_GAS_VRC_20.i_xClsLS <-> Channel 4/fb_AT1K0_GAS_VRC_20.i_xClsLS
//     PlcTask Inputs/GVL_Devices.fb_AT1K0_GAS_VRC_10.i_xOpnLS <-> Channel 1/fb_AT1K0_GAS_VRC_10.i_xOpnLS
//     PlcTask Inputs/GVL_Devices.fb_AT1K0_GAS_VRC_20.i_xOpnLS <-> Channel 3/fb_AT1K0_GAS_VRC_20.i_xOpnLS
//   plc_kfe_gatt Instance <-> =+-CX2020/EtherCAT1/=+-EK1100_02_00/=+-ES1004_02_04
//     PlcTask Inputs/GVL_Devices.fb_AT1K0_GAS_VRC_30.i_xClsLS <-> Channel 2/fb_AT1K0_GAS_VRC_30.i_xClsLS
//     PlcTask Inputs/GVL_Devices.fb_AT1K0_GAS_VRC_40.i_xClsLS <-> Channel 4/fb_AT1K0_GAS_VRC_40.i_xClsLS
//     PlcTask Inputs/GVL_Devices.fb_AT1K0_GAS_VRC_30.i_xOpnLS <-> Channel 1/fb_AT1K0_GAS_VRC_30.i_xOpnLS
//     PlcTask Inputs/GVL_Devices.fb_AT1K0_GAS_VRC_40.i_xOpnLS <-> Channel 3/fb_AT1K0_GAS_VRC_40.i_xOpnLS
//   plc_kfe_gatt Instance <-> =+-CX2020/EtherCAT1/=+-EK1100_02_00/=+-ES1004_02_08
//     PlcTask Inputs/GVL_Devices.fb_AT1K0_GAS_VRC_50.i_xClsLS <-> Channel 2/Input
//     PlcTask Inputs/GVL_Devices.fb_AT1K0_GAS_VRC_60.i_xClsLS <-> Channel 4/Input
//     PlcTask Inputs/GVL_Devices.fb_AT1K0_GAS_VRC_50.i_xOpnLS <-> Channel 1/Input
//     PlcTask Inputs/GVL_Devices.fb_AT1K0_GAS_VRC_60.i_xOpnLS <-> Channel 3/Input
//   plc_kfe_gatt Instance <-> =+-CX2020/EtherCAT1/=+-EK1100_02_00/=+-ES2004_02_01
//     PlcTask Outputs/GVL_Devices.fb_AT1K0_GAS_VRC_10.q_xOPN_DO <-> Channel 1/fb_AT1K0_GAS_VRC_10.q_xOPN_DO
//     PlcTask Outputs/GVL_Devices.fb_AT1K0_GAS_VRC_20.q_xOPN_DO <-> Channel 3/fb_AT1K0_GAS_VRC_20.q_xOPN_DO
//     PlcTask Outputs/GVL_Devices.fb_AT1K0_GAS_VRC_10.q_xOPN_DO_2 <-> Channel 2/fb_AT1K0_GAS_VRC_10.q_xOPN_DO
//     PlcTask Outputs/GVL_Devices.fb_AT1K0_GAS_VRC_20.q_xOPN_DO_2 <-> Channel 4/fb_AT1K0_GAS_VRC_20.q_xOPN_DO
//   plc_kfe_gatt Instance <-> =+-CX2020/EtherCAT1/=+-EK1100_02_00/=+-ES2004_02_03
//     PlcTask Outputs/GVL_Devices.fb_AT1K0_GAS_VRC_30.q_xOPN_DO <-> Channel 1/fb_AT1K0_GAS_VRC_30.q_xOPN_DO
//     PlcTask Outputs/GVL_Devices.fb_AT1K0_GAS_VRC_40.q_xOPN_DO <-> Channel 3/fb_AT1K0_GAS_VRC_40.q_xOPN_DO
//     PlcTask Outputs/GVL_Devices.fb_AT1K0_GAS_VRC_30.q_xOPN_DO_2 <-> Channel 2/fb_AT1K0_GAS_VRC_30.q_xOPN_DO
//     PlcTask Outputs/GVL_Devices.fb_AT1K0_GAS_VRC_40.q_xOPN_DO_2 <-> Channel 4/fb_AT1K0_GAS_VRC_40.q_xOPN_DO
//   plc_kfe_gatt Instance <-> =+-CX2020/EtherCAT1/=+-EK1100_02_00/=+-ES2004_02_07
//     PlcTask Outputs/GVL_Devices.fb_AT1K0_GAS_VRC_50.q_xOPN_DO <-> Channel 1/Output
//     PlcTask Outputs/GVL_Devices.fb_AT1K0_GAS_VRC_60.q_xOPN_DO <-> Channel 2/Output
//     PlcTask Outputs/Main.M2.bBrakeRelease <-> Channel 3/Output
//     PlcTask Outputs/Main.M4.bBrakeRelease <-> Channel 4/Output
//   plc_kfe_gatt Instance <-> =+-CX2020/EtherCAT1/=+-EK1100_02_00/=+-ES7041_02_05
//     PlcTask Inputs/Main.M1.bLimitBackwardEnable <-> STM Status/Status/Digital input 2
//     PlcTask Inputs/Main.M1.bLimitForwardEnable <-> STM Status/Status/Digital input 1
//   plc_kfe_gatt Instance <-> =+-CX2020/EtherCAT1/=+-EK1100_02_00/=+-ES7041_02_06
//     PlcTask Inputs/Main.M2.bLimitBackwardEnable <-> STM Status/Status/Digital input 1
//     PlcTask Inputs/Main.M2.bLimitForwardEnable <-> STM Status/Status/Digital input 2
//   plc_kfe_gatt Instance <-> =+-CX2020/EtherCAT1/=+-EK1100_02_00/=+-ES7041_02_09
//     PlcTask Inputs/Main.M3.bLimitBackwardEnable <-> STM Status/Status/Digital input 2
//     PlcTask Inputs/Main.M3.bLimitForwardEnable <-> STM Status/Status/Digital input 1
//   plc_kfe_gatt Instance <-> =+-CX2020/EtherCAT1/=+-EK1100_02_00/=+-ES7041_02_10
//     PlcTask Inputs/Main.M4.bLimitBackwardEnable <-> STM Status/Status/Digital input 1
//     PlcTask Inputs/Main.M4.bLimitForwardEnable <-> STM Status/Status/Digital input 2
//   plc_kfe_gatt Instance <-> =+-CX2020/EtherCAT1/=+-EK1100_03_00/=+-EL2798_03_03
//     PlcTask Outputs/GVL_Devices.fb_AT1K0_GAS_PTM_10.q_xProtection <-> Channel 4/fb_AT1K0_GAS_PTM_10.q_xProtection
//     PlcTask Outputs/GVL_Devices.fb_AT1K0_GAS_PTM_10.q_xReset <-> Channel 1/fb_AT1K0_GAS_PTM_10.q_xReset
//     PlcTask Outputs/GVL_Devices.fb_AT1K0_GAS_PTM_10.q_xSetSpeed <-> Channel 5/fb_AT1K0_GAS_PTM_10.q_xSetSpeed
//     PlcTask Outputs/GVL_Devices.fb_AT1K0_GAS_PTM_10.q_xStart <-> Channel 2/fb_AT1K0_GAS_PTM_10.q_xStart
//     PlcTask Outputs/GVL_Devices.fb_AT1K0_GAS_PTM_10.q_xStop <-> Channel 3/fb_AT1K0_GAS_PTM_10.q_xStop
//   plc_kfe_gatt Instance <-> =+-CX2020/EtherCAT1/=+-EK1100_03_00/=+-EL2798_03_07
//     PlcTask Outputs/GVL_Devices.fb_AT1K0_GAS_PTM_20.q_xProtection <-> Channel 4/fb_AT1K0_GAS_PTM_20.q_xProtection
//     PlcTask Outputs/GVL_Devices.fb_AT1K0_GAS_PTM_20.q_xReset <-> Channel 1/fb_AT1K0_GAS_PTM_20.q_xReset
//     PlcTask Outputs/GVL_Devices.fb_AT1K0_GAS_PTM_20.q_xSetSpeed <-> Channel 5/fb_AT1K0_GAS_PTM_20.q_xSetSpeed
//     PlcTask Outputs/GVL_Devices.fb_AT1K0_GAS_PTM_20.q_xStart <-> Channel 2/fb_AT1K0_GAS_PTM_20.q_xStart
//     PlcTask Outputs/GVL_Devices.fb_AT1K0_GAS_PTM_20.q_xStop <-> Channel 3/fb_AT1K0_GAS_PTM_20.q_xStop
//   plc_kfe_gatt Instance <-> =+-CX2020/EtherCAT1/=+-EK1100_03_00/=+-EL2798_03_13
//     PlcTask Outputs/GVL_Devices.fb_AT1K0_GAS_PTM_30.q_xProtection <-> Channel 4/fb_AT1K0_GAS_PTM_30.q_xProtection
//     PlcTask Outputs/GVL_Devices.fb_AT1K0_GAS_PTM_30.q_xReset <-> Channel 1/fb_AT1K0_GAS_PTM_30.q_xReset
//     PlcTask Outputs/GVL_Devices.fb_AT1K0_GAS_PTM_30.q_xSetSpeed <-> Channel 5/fb_AT1K0_GAS_PTM_30.q_xSetSpeed
//     PlcTask Outputs/GVL_Devices.fb_AT1K0_GAS_PTM_30.q_xStart <-> Channel 2/fb_AT1K0_GAS_PTM_30.q_xStart
//     PlcTask Outputs/GVL_Devices.fb_AT1K0_GAS_PTM_30.q_xStop <-> Channel 3/fb_AT1K0_GAS_PTM_30.q_xStop
//   plc_kfe_gatt Instance <-> =+-CX2020/EtherCAT1/=+-EK1100_03_00/=+-EL2798_03_17
//     PlcTask Outputs/GVL_Devices.fb_AT1K0_GAS_PTM_40.q_xProtection <-> Channel 4/fb_AT1K0_GAS_PTM_40.q_xProtection
//     PlcTask Outputs/GVL_Devices.fb_AT1K0_GAS_PTM_40.q_xReset <-> Channel 1/fb_AT1K0_GAS_PTM_40.q_xReset
//     PlcTask Outputs/GVL_Devices.fb_AT1K0_GAS_PTM_40.q_xSetSpeed <-> Channel 5/fb_AT1K0_GAS_PTM_40.q_xSetSpeed
//     PlcTask Outputs/GVL_Devices.fb_AT1K0_GAS_PTM_40.q_xStart <-> Channel 2/fb_AT1K0_GAS_PTM_40.q_xStart
//     PlcTask Outputs/GVL_Devices.fb_AT1K0_GAS_PTM_40.q_xStop <-> Channel 3/fb_AT1K0_GAS_PTM_40.q_xStop
//   plc_kfe_gatt Instance <-> =+-CX2020/EtherCAT1/=+-EK1100_03_00/=+-ES1004_03_01
//     PlcTask Inputs/GVL_Devices.fb_AT1K0_GAS_PTM_10.i_xAtSpd <-> Channel 2/fb_AT1K0_GAS_PTM_10.i_xAtSpd
//     PlcTask Inputs/GVL_Devices.fb_AT1K0_GAS_PTM_10.i_xDecel <-> Channel 1/fb_AT1K0_GAS_PTM_10.i_xDecel
//     PlcTask Inputs/GVL_Devices.fb_AT1K0_GAS_PTM_10.i_xNCFault <-> Channel 3/fb_AT1K0_GAS_PTM_10.i_xNCFault
//     PlcTask Inputs/GVL_Devices.fb_AT1K0_GAS_PTM_10.i_xRotate <-> Channel 4/fb_AT1K0_GAS_PTM_10.i_xRotate
//   plc_kfe_gatt Instance <-> =+-CX2020/EtherCAT1/=+-EK1100_03_00/=+-ES1004_03_02
//     PlcTask Inputs/GVL_Devices.fb_AT1K0_GAS_PTM_10.i_xAccel <-> Channel 1/fb_AT1K0_GAS_PTM_10.i_xAccel
//   plc_kfe_gatt Instance <-> =+-CX2020/EtherCAT1/=+-EK1100_03_00/=+-ES1004_03_08
//     PlcTask Inputs/GVL_Devices.fb_AT1K0_GAS_PTM_20.i_xAtSpd <-> Channel 2/fb_AT1K0_GAS_PTM_20.i_xAtSpd
//     PlcTask Inputs/GVL_Devices.fb_AT1K0_GAS_PTM_20.i_xDecel <-> Channel 1/fb_AT1K0_GAS_PTM_20.i_xDecel
//     PlcTask Inputs/GVL_Devices.fb_AT1K0_GAS_PTM_20.i_xNCFault <-> Channel 3/fb_AT1K0_GAS_PTM_20.i_xNCFault
//     PlcTask Inputs/GVL_Devices.fb_AT1K0_GAS_PTM_20.i_xRotate <-> Channel 4/fb_AT1K0_GAS_PTM_20.i_xRotate
//   plc_kfe_gatt Instance <-> =+-CX2020/EtherCAT1/=+-EK1100_03_00/=+-ES1004_03_09
//     PlcTask Inputs/GVL_Devices.fb_AT1K0_GAS_PTM_20.i_xAccel <-> Channel 1/fb_AT1K0_GAS_PTM_20.i_xAccel
//   plc_kfe_gatt Instance <-> =+-CX2020/EtherCAT1/=+-EK1100_03_00/=+-ES1004_03_11
//     PlcTask Inputs/GVL_Devices.fb_AT1K0_GAS_PTM_30.i_xAtSpd <-> Channel 2/fb_AT1K0_GAS_PTM_30.i_xAtSpd
//     PlcTask Inputs/GVL_Devices.fb_AT1K0_GAS_PTM_30.i_xDecel <-> Channel 1/fb_AT1K0_GAS_PTM_30.i_xDecel
//     PlcTask Inputs/GVL_Devices.fb_AT1K0_GAS_PTM_30.i_xNCFault <-> Channel 3/fb_AT1K0_GAS_PTM_30.i_xNCFault
//     PlcTask Inputs/GVL_Devices.fb_AT1K0_GAS_PTM_30.i_xRotate <-> Channel 4/fb_AT1K0_GAS_PTM_30.i_xRotate
//   plc_kfe_gatt Instance <-> =+-CX2020/EtherCAT1/=+-EK1100_03_00/=+-ES1004_03_12
//     PlcTask Inputs/GVL_Devices.fb_AT1K0_GAS_PTM_30.i_xAccel <-> Channel 1/fb_AT1K0_GAS_PTM_30.i_xAccel
//   plc_kfe_gatt Instance <-> =+-CX2020/EtherCAT1/=+-EK1100_03_00/=+-ES1004_03_18
//     PlcTask Inputs/GVL_Devices.fb_AT1K0_GAS_PTM_40.i_xAtSpd <-> Channel 2/fb_AT1K0_GAS_PTM_40.i_xAtSpd
//     PlcTask Inputs/GVL_Devices.fb_AT1K0_GAS_PTM_40.i_xDecel <-> Channel 1/fb_AT1K0_GAS_PTM_40.i_xDecel
//     PlcTask Inputs/GVL_Devices.fb_AT1K0_GAS_PTM_40.i_xNCFault <-> Channel 3/fb_AT1K0_GAS_PTM_40.i_xNCFault
//     PlcTask Inputs/GVL_Devices.fb_AT1K0_GAS_PTM_40.i_xRotate <-> Channel 4/fb_AT1K0_GAS_PTM_40.i_xRotate
//   plc_kfe_gatt Instance <-> =+-CX2020/EtherCAT1/=+-EK1100_03_00/=+-ES1004_03_19
//     PlcTask Inputs/GVL_Devices.fb_AT1K0_GAS_PTM_40.i_xAccel <-> Channel 1/fb_AT1K0_GAS_PTM_40.i_xAccel
//   plc_kfe_gatt Instance <-> =+-CX2020/EtherCAT1/=+-EK1100_03_00/=+-ES3064_03_04
//     PlcTask Inputs/GVL_Devices.fb_AT1K0_GAS_PTM_10.i_iCurrentMon <-> AI Standard Channel 2/fb_AT1K0_GAS_PTM_10.i_iCurrentMon
//     PlcTask Inputs/GVL_Devices.fb_AT1K0_GAS_PTM_10.i_iRawSpeed <-> AI Standard Channel 1/fb_AT1K0_GAS_PTM_10.i_iRawSpeed
//     PlcTask Inputs/GVL_Devices.fb_AT1K0_GAS_PTM_10.i_iTempMon <-> AI Standard Channel 3/fb_AT1K0_GAS_PTM_10.i_iTempMon
//   plc_kfe_gatt Instance <-> =+-CX2020/EtherCAT1/=+-EK1100_03_00/=+-ES3064_03_06
//     PlcTask Inputs/GVL_Devices.fb_AT1K0_GAS_PTM_20.i_iCurrentMon <-> AI Standard Channel 2/fb_AT1K0_GAS_PTM_20.i_iCurrentMon
//     PlcTask Inputs/GVL_Devices.fb_AT1K0_GAS_PTM_20.i_iRawSpeed <-> AI Standard Channel 1/fb_AT1K0_GAS_PTM_20.i_iRawSpeed
//     PlcTask Inputs/GVL_Devices.fb_AT1K0_GAS_PTM_20.i_iTempMon <-> AI Standard Channel 3/fb_AT1K0_GAS_PTM_20.i_iTempMon
//   plc_kfe_gatt Instance <-> =+-CX2020/EtherCAT1/=+-EK1100_03_00/=+-ES3064_03_14
//     PlcTask Inputs/GVL_Devices.fb_AT1K0_GAS_PTM_30.i_iCurrentMon <-> AI Standard Channel 2/fb_AT1K0_GAS_PTM_30.i_iCurrentMon
//     PlcTask Inputs/GVL_Devices.fb_AT1K0_GAS_PTM_30.i_iRawSpeed <-> AI Standard Channel 1/fb_AT1K0_GAS_PTM_30.i_iRawSpeed
//     PlcTask Inputs/GVL_Devices.fb_AT1K0_GAS_PTM_30.i_iTempMon <-> AI Standard Channel 3/fb_AT1K0_GAS_PTM_30.i_iTempMon
//   plc_kfe_gatt Instance <-> =+-CX2020/EtherCAT1/=+-EK1100_03_00/=+-ES3064_03_16
//     PlcTask Inputs/GVL_Devices.fb_AT1K0_GAS_PTM_40.i_iCurrentMon <-> AI Standard Channel 2/fb_AT1K0_GAS_PTM_40.i_iCurrentMon
//     PlcTask Inputs/GVL_Devices.fb_AT1K0_GAS_PTM_40.i_iRawSpeed <-> AI Standard Channel 1/fb_AT1K0_GAS_PTM_40.i_iRawSpeed
//     PlcTask Inputs/GVL_Devices.fb_AT1K0_GAS_PTM_40.i_iTempMon <-> AI Standard Channel 3/fb_AT1K0_GAS_PTM_40.i_iTempMon
//   plc_kfe_gatt Instance <-> =+-CX2020/EtherCAT1/=+-EK1100_03_00/=+-ES4004_03_05
//     PlcTask Outputs/GVL_Devices.fb_AT1K0_GAS_PTM_10.q_iSpeedSet <-> AO Outputs Channel 1/fb_AT1K0_GAS_PTM_10.q_iSpeedSet
//     PlcTask Outputs/GVL_Devices.fb_AT1K0_GAS_PTM_20.q_iSpeedSet <-> AO Outputs Channel 3/fb_AT1K0_GAS_PTM_20.q_iSpeedSet
//   plc_kfe_gatt Instance <-> =+-CX2020/EtherCAT1/=+-EK1100_03_00/=+-ES4004_03_15
//     PlcTask Outputs/GVL_Devices.fb_AT1K0_GAS_PTM_30.q_iSpeedSet <-> AO Outputs Channel 1/fb_AT1K0_GAS_PTM_30.q_iSpeedSet
//     PlcTask Outputs/GVL_Devices.fb_AT1K0_GAS_PTM_40.q_iSpeedSet <-> AO Outputs Channel 3/fb_AT1K0_GAS_PTM_40.q_iSpeedSet
//   plc_kfe_gatt Instance <-> =+-CX2020/EtherCAT1/=+-EK1100_04_00/=+-EL3174_04_17
//     PlcTask Inputs/GVL_Devices.GCM_70.i_iPRESS_R <-> AI Standard Channel 3/GCM_70.i_iPRESS_R
//     PlcTask Inputs/GVL_Devices.GCM_80.i_iPRESS_R <-> AI Standard Channel 1/GCM_80.i_iPRESS_R
//     PlcTask Inputs/GVL_Devices.GCM_81.i_iPRESS_R <-> AI Standard Channel 2/Value
//   plc_kfe_gatt Instance <-> =+-CX2020/EtherCAT1/=+-EK1100_04_00/=+-EL7041_04_07
//     PlcTask Inputs/Main.M5.bLimitBackwardEnable <-> STM Status/Status/Digital input 1
//     PlcTask Inputs/Main.M5.bLimitForwardEnable <-> STM Status/Status/Digital input 2
//   plc_kfe_gatt Instance <-> =+-CX2020/EtherCAT1/=+-EK1100_04_00/=+-EL7041_04_08
//     PlcTask Inputs/Main.M6.bLimitBackwardEnable <-> STM Status/Status/Digital input 1
//     PlcTask Inputs/Main.M6.bLimitForwardEnable <-> STM Status/Status/Digital input 2
//   plc_kfe_gatt Instance <-> =+-CX2020/EtherCAT1/=+-EK1100_04_00/=+-EL7041_04_10
//     PlcTask Inputs/Main.M7.bLimitBackwardEnable <-> STM Status/Status/Digital input 1
//     PlcTask Inputs/Main.M7.bLimitForwardEnable <-> STM Status/Status/Digital input 2
//   plc_kfe_gatt Instance <-> =+-CX2020/EtherCAT1/=+-EK1100_04_00/=+-EL7041_04_11
//     PlcTask Inputs/Main.M8.bLimitBackwardEnable <-> STM Status/Status/Digital input 1
//     PlcTask Inputs/Main.M8.bLimitForwardEnable <-> STM Status/Status/Digital input 2
//   plc_kfe_gatt Instance <-> =+-CX2020/EtherCAT1/=+-EK1100_04_00/=+-ES1084_04_06
//     PlcTask Inputs/GVL_Devices.fb_AT1K0_GAS_PTM_80.i_xAtSpd <-> Channel 1/fb_AT1K0_GAS_PTM_80.i_xAtSpd
//     PlcTask Inputs/GVL_Devices.fb_AT1K0_GAS_PTM_80.i_xFault <-> Channel 2/fb_AT1K0_GAS_PTM_80.i_xFault
//   plc_kfe_gatt Instance <-> =+-CX2020/EtherCAT1/=+-EK1100_04_00/=+-ES2004_04_01
//     PlcTask Outputs/GVL_Devices.VVC_71.q_xOPN_DO <-> Channel 1/VVC_71.q_xOPN_DO
//     PlcTask Outputs/GVL_Devices.VVC_72.q_xOPN_DO <-> Channel 2/VVC_72.q_xOPN_DO
//     PlcTask Outputs/GVL_Devices.fb_AT1K0_GAS_PTM_80.q_RunDO <-> Channel 3/fb_AT1K0_GAS_PTM_80.q_RunDO
//   plc_kfe_gatt Instance <-> =+-CX2020/EtherCAT1/=+-EK1100_04_00/=+-ES2004_04_09
//     PlcTask Outputs/Main.M{5..8}.bBrakeRelease <-> Channel {1..4}/Output  (4 links)
//   plc_kfe_gatt Instance <-> =+-CX2020/EtherCAT1/=+-EK1100_04_00/=+-ES4004_04_02
//     PlcTask Outputs/GVL_Devices.VCN_70.q_iRawPosition <-> AO Outputs Channel 1/VCN_70.q_iRawPosition
//   plc_kfe_gatt Instance <-> =+-CX2020/EtherCAT1/=+-EK1100_05_00/=+-EL1084_05_12
//     PlcTask Inputs/GVL_Devices.fb_AT1K0_GAS_PMF_110.i_xAlarmOK <-> Channel 2/fb_AT1K0_GAS_PMF_110.i_xAlarmOK
//     PlcTask Inputs/GVL_Devices.fb_AT1K0_GAS_PMF_120.i_xAlarmOK <-> Channel 4/fb_AT1K0_GAS_PMF_120.i_xAlarmOK
//     PlcTask Inputs/GVL_Devices.fb_AT1K0_GAS_PMF_110.i_xIsRun <-> Channel 1/fb_AT1K0_GAS_PMF_110.i_xIsRun
//     PlcTask Inputs/GVL_Devices.fb_AT1K0_GAS_PMF_120.i_xIsRun <-> Channel 3/fb_AT1K0_GAS_PMF_120.i_xIsRun
//   plc_kfe_gatt Instance <-> =+-CX2020/EtherCAT1/=+-EK1100_05_00/=+-EL1084_05_13
//     PlcTask Inputs/GVL_Devices.fb_AT1K0_GAS_PMF_140.i_xAlarmOK <-> Channel 2/fb_AT1K0_GAS_PMF_140.i_xAlarmOK
//     PlcTask Inputs/GVL_Devices.fb_AT1K0_GAS_PMF_140.i_xIsRun <-> Channel 1/fb_AT1K0_GAS_PMF_140.i_xIsRun
//   plc_kfe_gatt Instance <-> =+-CX2020/EtherCAT1/=+-EK1100_05_00/=+-EL2798_05_10
//     PlcTask Outputs/GVL_Devices.fb_AT1K0_GAS_PMF_110.q_xResetAlarm <-> Channel 2/fb_AT1K0_GAS_PMF_110.q_xResetAlarm
//     PlcTask Outputs/GVL_Devices.fb_AT1K0_GAS_PMF_120.q_xResetAlarm <-> Channel 4/fb_AT1K0_GAS_PMF_120.q_xResetAlarm
//     PlcTask Outputs/GVL_Devices.fb_AT1K0_GAS_PMF_140.q_xResetAlarm <-> Channel 6/fb_AT1K0_GAS_PMF_140.q_xResetAlarm
//     PlcTask Outputs/GVL_Devices.fb_AT1K0_GAS_PMF_110.q_xRunDo <-> Channel 1/fb_AT1K0_GAS_PMF_110.q_xRunDo
//     PlcTask Outputs/GVL_Devices.fb_AT1K0_GAS_PMF_120.q_xRunDo <-> Channel 3/fb_AT1K0_GAS_PMF_120.q_xRunDo
//     PlcTask Outputs/GVL_Devices.fb_AT1K0_GAS_PMF_140.q_xRunDo <-> Channel 5/fb_AT1K0_GAS_PMF_140.q_xRunDo
//   plc_kfe_gatt Instance <-> =+-CX2020/EtherCAT1/=+-EK1100_05_00/=+-EL3174_05_16
//     PlcTask Inputs/GVL_Devices.fb_AT1K0_GAS_GPI_111.i_iPRESS_R <-> AI Standard Channel 1/fb_AT1K0_GAS_GPI_111.i_iPRESS_R
//     PlcTask Inputs/GVL_Devices.fb_AT1K0_GAS_GPI_141.i_iPRESS_R <-> AI Standard Channel 3/fb_AT1K0_GAS_GPI_141.i_iPRESS_R
//     PlcTask Inputs/GVL_Devices.fb_AT1K0_GAS_GPI_121.i_iPRESS_R <-> AI Standard Channel 2/Value
//   plc_kfe_gatt Instance <-> =+-CX2020/EtherCAT1/=+-EK1100_05_00/=+-ES1004_05_01
//     PlcTask Inputs/GVL_Devices.fb_AT1K0_GAS_VRC_70.i_xClsLS <-> Channel 2/fb_AT1K0_GAS_VRC_70.i_xClsLS
//     PlcTask Inputs/GVL_Devices.fb_AT1K0_GAS_VRC_80.i_xClsLS <-> Channel 4/fb_AT1K0_GAS_VRC_80.i_xClsLS
//     PlcTask Inputs/GVL_Devices.fb_AT1K0_GAS_VRC_70.i_xOpnLS <-> Channel 1/fb_AT1K0_GAS_VRC_70.i_xOpnLS
//     PlcTask Inputs/GVL_Devices.fb_AT1K0_GAS_VRC_80.i_xOpnLS <-> Channel 3/fb_AT1K0_GAS_VRC_80.i_xOpnLS
//   plc_kfe_gatt Instance <-> =+-CX2020/EtherCAT1/=+-EK1100_05_00/=+-ES1004_05_03
//     PlcTask Inputs/GVL_Devices.fb_AT1K0_GAS_VRC_100.i_xClsLS <-> Channel 4/fb_AT1K0_GAS_VRC_100.i_xClsLS
//     PlcTask Inputs/GVL_Devices.fb_AT1K0_GAS_VRC_90.i_xClsLS <-> Channel 2/fb_AT1K0_GAS_VRC_90.i_xClsLS
//     PlcTask Inputs/GVL_Devices.fb_AT1K0_GAS_VRC_100.i_xOpnLS <-> Channel 3/fb_AT1K0_GAS_VRC_100.i_xOpnLS
//     PlcTask Inputs/GVL_Devices.fb_AT1K0_GAS_VRC_90.i_xOpnLS <-> Channel 1/fb_AT1K0_GAS_VRC_90.i_xOpnLS
//   plc_kfe_gatt Instance <-> =+-CX2020/EtherCAT1/=+-EK1100_05_00/=+-ES1004_05_06
//     PlcTask Inputs/GVL_Devices.fb_AT1K0_GAS_VRC_110.i_xClsLS <-> Channel 2/fb_AT1K0_GAS_VRC_110.i_xClsLS
//     PlcTask Inputs/GVL_Devices.fb_AT1K0_GAS_VRC_120.i_xClsLS <-> Channel 4/fb_AT1K0_GAS_VRC_120.i_xClsLS
//     PlcTask Inputs/GVL_Devices.fb_AT1K0_GAS_VRC_110.i_xOpnLS <-> Channel 1/fb_AT1K0_GAS_VRC_110.i_xOpnLS
//     PlcTask Inputs/GVL_Devices.fb_AT1K0_GAS_VRC_120.i_xOpnLS <-> Channel 3/fb_AT1K0_GAS_VRC_120.i_xOpnLS
//   plc_kfe_gatt Instance <-> =+-CX2020/EtherCAT1/=+-EK1100_05_00/=+-ES1004_05_08
//     PlcTask Inputs/GVL_Devices.fb_AT1K0_GAS_VRC_130.i_xClsLS <-> Channel 2/fb_AT1K0_GAS_VRC_130.i_xClsLS
//     PlcTask Inputs/GVL_Devices.fb_AT1K0_GAS_VRC_140.i_xClsLS <-> Channel 4/fb_AT1K0_GAS_VRC_140.i_xClsLS
//     PlcTask Inputs/GVL_Devices.fb_AT1K0_GAS_VRC_130.i_xOpnLS <-> Channel 1/fb_AT1K0_GAS_VRC_130.i_xOpnLS
//     PlcTask Inputs/GVL_Devices.fb_AT1K0_GAS_VRC_140.i_xOpnLS <-> Channel 3/fb_AT1K0_GAS_VRC_140.i_xOpnLS
//   plc_kfe_gatt Instance <-> =+-CX2020/EtherCAT1/=+-EK1100_05_00/=+-ES2004_05_02
//     PlcTask Outputs/GVL_Devices.fb_AT1K0_GAS_VRC_70.q_xOPN_DO <-> Channel 1/fb_AT1K0_GAS_VRC_70.q_xOPN_DO
//     PlcTask Outputs/GVL_Devices.fb_AT1K0_GAS_VRC_80.q_xOPN_DO <-> Channel 2/fb_AT1K0_GAS_VRC_80.q_xOPN_DO
//   plc_kfe_gatt Instance <-> =+-CX2020/EtherCAT1/=+-EK1100_05_00/=+-ES2004_05_04
//     PlcTask Outputs/GVL_Devices.fb_AT1K0_GAS_VRC_100.q_xOPN_DO <-> Channel 2/fb_AT1K0_GAS_VRC_100.q_xOPN_DO
//     PlcTask Outputs/GVL_Devices.fb_AT1K0_GAS_VRC_90.q_xOPN_DO <-> Channel 1/fb_AT1K0_GAS_VRC_90.q_xOPN_DO
//   plc_kfe_gatt Instance <-> =+-CX2020/EtherCAT1/=+-EK1100_05_00/=+-ES2004_05_05
//     PlcTask Outputs/GVL_Devices.fb_AT1K0_GAS_VRC_110.q_xOPN_DO <-> Channel 1/fb_AT1K0_GAS_VRC_110.q_xOPN_DO
//     PlcTask Outputs/GVL_Devices.fb_AT1K0_GAS_VRC_120.q_xOPN_DO <-> Channel 2/fb_AT1K0_GAS_VRC_120.q_xOPN_DO
//   plc_kfe_gatt Instance <-> =+-CX2020/EtherCAT1/=+-EK1100_05_00/=+-ES2004_05_07
//     PlcTask Outputs/GVL_Devices.fb_AT1K0_GAS_VRC_130.q_xOPN_DO <-> Channel 1/fb_AT1K0_GAS_VRC_130.q_xOPN_DO
//     PlcTask Outputs/GVL_Devices.fb_AT1K0_GAS_VRC_140.q_xOPN_DO <-> Channel 2/fb_AT1K0_GAS_VRC_140.q_xOPN_DO
//   plc_kfe_gatt Instance <-> =+-CX2020/EtherCAT1/=+-EK1100_06_00/=+-EL2794_06_22
//     PlcTask Outputs/GVL_Devices.fb_AT1K0_GAS_PMF_100.q_xBPStart <-> Channel 4/fb_AT1K0_GAS_PMF_100.q_xBPStart
//     PlcTask Outputs/GVL_Devices.fb_AT1K0_GAS_PMF_90.q_xBPStart <-> Channel 2/fb_AT1K0_GAS_PMF_90.q_xBPStart
//     PlcTask Outputs/GVL_Devices.fb_AT1K0_GAS_PMF_100.q_xMPStart <-> Channel 3/fb_AT1K0_GAS_PMF_100.q_xMPStart
//     PlcTask Outputs/GVL_Devices.fb_AT1K0_GAS_PMF_90.q_xMPStart <-> Channel 1/fb_AT1K0_GAS_PMF_90.q_xMPStart
//   plc_kfe_gatt Instance <-> =+-CX2020/EtherCAT1/=+-EK1100_06_00/=+-EL2798_06_03
//     PlcTask Outputs/GVL_Devices.fb_AT1K0_GAS_PTM_110.q_xProtection <-> Channel 5/fb_AT1K0_GAS_PTM_110.q_xProtection
//     PlcTask Outputs/GVL_Devices.fb_AT1K0_GAS_PTM_110.q_xReset <-> Channel 1/fb_AT1K0_GAS_PTM_110.q_xReset
//     PlcTask Outputs/GVL_Devices.fb_AT1K0_GAS_PTM_110.q_xSetSpeed <-> Channel 4/fb_AT1K0_GAS_PTM_110.q_xSetSpeed
//     PlcTask Outputs/GVL_Devices.fb_AT1K0_GAS_PTM_110.q_xStart <-> Channel 2/fb_AT1K0_GAS_PTM_110.q_xStart
//     PlcTask Outputs/GVL_Devices.fb_AT1K0_GAS_PTM_110.q_xStop <-> Channel 3/fb_AT1K0_GAS_PTM_110.q_xStop
//   plc_kfe_gatt Instance <-> =+-CX2020/EtherCAT1/=+-EK1100_06_00/=+-EL2798_06_07
//     PlcTask Outputs/GVL_Devices.fb_AT1K0_GAS_PTM_120.q_xProtection <-> Channel 4/fb_AT1K0_GAS_PTM_120.q_xProtection
//     PlcTask Outputs/GVL_Devices.fb_AT1K0_GAS_PTM_120.q_xReset <-> Channel 1/fb_AT1K0_GAS_PTM_120.q_xReset
//     PlcTask Outputs/GVL_Devices.fb_AT1K0_GAS_PTM_120.q_xSetSpeed <-> Channel 5/fb_AT1K0_GAS_PTM_120.q_xSetSpeed
//     PlcTask Outputs/GVL_Devices.fb_AT1K0_GAS_PTM_120.q_xStart <-> Channel 2/fb_AT1K0_GAS_PTM_120.q_xStart
//     PlcTask Outputs/GVL_Devices.fb_AT1K0_GAS_PTM_120.q_xStop <-> Channel 3/fb_AT1K0_GAS_PTM_120.q_xStop
//   plc_kfe_gatt Instance <-> =+-CX2020/EtherCAT1/=+-EK1100_06_00/=+-EL2798_06_13
//     PlcTask Outputs/GVL_Devices.fb_AT1K0_GAS_PTM_130.q_xProtection <-> Channel 4/fb_AT1K0_GAS_PTM_130.q_xProtection
//     PlcTask Outputs/GVL_Devices.fb_AT1K0_GAS_PTM_130.q_xReset <-> Channel 1/fb_AT1K0_GAS_PTM_130.q_xReset
//     PlcTask Outputs/GVL_Devices.fb_AT1K0_GAS_PTM_130.q_xSetSpeed <-> Channel 5/fb_AT1K0_GAS_PTM_130.q_xSetSpeed
//     PlcTask Outputs/GVL_Devices.fb_AT1K0_GAS_PTM_130.q_xStart <-> Channel 2/fb_AT1K0_GAS_PTM_130.q_xStart
//     PlcTask Outputs/GVL_Devices.fb_AT1K0_GAS_PTM_130.q_xStop <-> Channel 3/fb_AT1K0_GAS_PTM_130.q_xStop
//   plc_kfe_gatt Instance <-> =+-CX2020/EtherCAT1/=+-EK1100_06_00/=+-EL2798_06_17
//     PlcTask Outputs/GVL_Devices.fb_AT1K0_GAS_PTM_140.q_xProtection <-> Channel 4/fb_AT1K0_GAS_PTM_140.q_xProtection
//     PlcTask Outputs/GVL_Devices.fb_AT1K0_GAS_PTM_140.q_xReset <-> Channel 1/fb_AT1K0_GAS_PTM_140.q_xReset
//     PlcTask Outputs/GVL_Devices.fb_AT1K0_GAS_PTM_140.q_xSetSpeed <-> Channel 5/fb_AT1K0_GAS_PTM_140.q_xSetSpeed
//     PlcTask Outputs/GVL_Devices.fb_AT1K0_GAS_PTM_140.q_xStart <-> Channel 2/fb_AT1K0_GAS_PTM_140.q_xStart
//     PlcTask Outputs/GVL_Devices.fb_AT1K0_GAS_PTM_140.q_xStop <-> Channel 3/fb_AT1K0_GAS_PTM_140.q_xStop
//   plc_kfe_gatt Instance <-> =+-CX2020/EtherCAT1/=+-EK1100_06_00/=+-ES1004_06_01
//     PlcTask Inputs/GVL_Devices.fb_AT1K0_GAS_PTM_110.i_xAccel <-> Channel 4/fb_AT1K0_GAS_PTM_110.i_xAccel
//     PlcTask Inputs/GVL_Devices.fb_AT1K0_GAS_PTM_110.i_xAtSpd <-> Channel 1/fb_AT1K0_GAS_PTM_110.i_xAtSpd
//     PlcTask Inputs/GVL_Devices.fb_AT1K0_GAS_PTM_110.i_xFaultNC <-> Channel 2/fb_AT1K0_GAS_PTM_110.i_xFaultNC
//     PlcTask Inputs/GVL_Devices.fb_AT1K0_GAS_PTM_110.i_xRotate <-> Channel 3/fb_AT1K0_GAS_PTM_110.i_xRotate
//   plc_kfe_gatt Instance <-> =+-CX2020/EtherCAT1/=+-EK1100_06_00/=+-ES1004_06_02
//     PlcTask Inputs/GVL_Devices.fb_AT1K0_GAS_PTM_110.i_xDecel <-> Channel 1/fb_AT1K0_GAS_PTM_110.i_xDecel
//   plc_kfe_gatt Instance <-> =+-CX2020/EtherCAT1/=+-EK1100_06_00/=+-ES1004_06_08
//     PlcTask Inputs/GVL_Devices.fb_AT1K0_GAS_PTM_120.i_xAtSpd <-> Channel 2/fb_AT1K0_GAS_PTM_120.i_xAtSpd
//     PlcTask Inputs/GVL_Devices.fb_AT1K0_GAS_PTM_120.i_xDecel <-> Channel 1/fb_AT1K0_GAS_PTM_120.i_xDecel
//     PlcTask Inputs/GVL_Devices.fb_AT1K0_GAS_PTM_120.i_xNCFault <-> Channel 3/fb_AT1K0_GAS_PTM_120.i_xNCFault
//     PlcTask Inputs/GVL_Devices.fb_AT1K0_GAS_PTM_120.i_xRotate <-> Channel 4/fb_AT1K0_GAS_PTM_120.i_xRotate
//   plc_kfe_gatt Instance <-> =+-CX2020/EtherCAT1/=+-EK1100_06_00/=+-ES1004_06_09
//     PlcTask Inputs/GVL_Devices.fb_AT1K0_GAS_PTM_120.i_xAccel <-> Channel 1/fb_AT1K0_GAS_PTM_120.i_xAccel
//   plc_kfe_gatt Instance <-> =+-CX2020/EtherCAT1/=+-EK1100_06_00/=+-ES1004_06_11
//     PlcTask Inputs/GVL_Devices.fb_AT1K0_GAS_PTM_130.i_xAtSpd <-> Channel 2/fb_AT1K0_GAS_PTM_130.i_xAtSpd
//     PlcTask Inputs/GVL_Devices.fb_AT1K0_GAS_PTM_130.i_xDecel <-> Channel 1/fb_AT1K0_GAS_PTM_130.i_xDecel
//     PlcTask Inputs/GVL_Devices.fb_AT1K0_GAS_PTM_130.i_xNCFault <-> Channel 3/fb_AT1K0_GAS_PTM_130.i_xNCFault
//     PlcTask Inputs/GVL_Devices.fb_AT1K0_GAS_PTM_130.i_xRotate <-> Channel 4/fb_AT1K0_GAS_PTM_130.i_xRotate
//   plc_kfe_gatt Instance <-> =+-CX2020/EtherCAT1/=+-EK1100_06_00/=+-ES1004_06_12
//     PlcTask Inputs/GVL_Devices.fb_AT1K0_GAS_PTM_130.i_xAccel <-> Channel 1/fb_AT1K0_GAS_PTM_130.i_xAccel
//   plc_kfe_gatt Instance <-> =+-CX2020/EtherCAT1/=+-EK1100_06_00/=+-ES1004_06_18
//     PlcTask Inputs/GVL_Devices.fb_AT1K0_GAS_PTM_140.i_xAtSpd <-> Channel 2/fb_AT1K0_GAS_PTM_140.i_xAtSpd
//     PlcTask Inputs/GVL_Devices.fb_AT1K0_GAS_PTM_140.i_xDecel <-> Channel 1/fb_AT1K0_GAS_PTM_140.i_xDecel
//     PlcTask Inputs/GVL_Devices.fb_AT1K0_GAS_PTM_140.i_xNCFault <-> Channel 3/fb_AT1K0_GAS_PTM_140.i_xNCFault
//     PlcTask Inputs/GVL_Devices.fb_AT1K0_GAS_PTM_140.i_xRotate <-> Channel 4/fb_AT1K0_GAS_PTM_140.i_xRotate
//   plc_kfe_gatt Instance <-> =+-CX2020/EtherCAT1/=+-EK1100_06_00/=+-ES1004_06_19
//     PlcTask Inputs/GVL_Devices.fb_AT1K0_GAS_PTM_140.i_xAccel <-> Channel 1/fb_AT1K0_GAS_PTM_140.i_xAccel
//   plc_kfe_gatt Instance <-> =+-CX2020/EtherCAT1/=+-EK1100_06_00/=+-ES1088_06_20
//     PlcTask Inputs/GVL_Devices.fb_AT1K0_GAS_PMF_90.i_xAlarmOK <-> Channel 4/fb_AT1K0_GAS_PMF_90.i_xAlarmOK
//     PlcTask Inputs/GVL_Devices.fb_AT1K0_GAS_PMF_90.i_xBPStatus <-> Channel 2/fb_AT1K0_GAS_PMF_90.i_xBPStatus
//     PlcTask Inputs/GVL_Devices.fb_AT1K0_GAS_PMF_90.i_xMPStatus <-> Channel 1/fb_AT1K0_GAS_PMF_90.i_xMPStatus
//     PlcTask Inputs/GVL_Devices.fb_AT1K0_GAS_PMF_90.i_xRemote <-> Channel 5/fb_AT1K0_GAS_PMF_90.i_xRemote
//     PlcTask Inputs/GVL_Devices.fb_AT1K0_GAS_PMF_90.i_xWarning <-> Channel 3/fb_AT1K0_GAS_PMF_90.i_xWarning
//   plc_kfe_gatt Instance <-> =+-CX2020/EtherCAT1/=+-EK1100_06_00/=+-ES1088_06_23
//     PlcTask Inputs/GVL_Devices.fb_AT1K0_GAS_PMF_100.i_xAlarmOK <-> Channel 4/fb_AT1K0_GAS_PMF_100.i_xAlarmOK
//     PlcTask Inputs/GVL_Devices.fb_AT1K0_GAS_PMF_100.i_xBPStatus <-> Channel 2/fb_AT1K0_GAS_PMF_100.i_xBPStatus
//     PlcTask Inputs/GVL_Devices.fb_AT1K0_GAS_PMF_100.i_xMPStatus <-> Channel 1/fb_AT1K0_GAS_PMF_100.i_xMPStatus
//     PlcTask Inputs/GVL_Devices.fb_AT1K0_GAS_PMF_100.i_xRemote <-> Channel 5/fb_AT1K0_GAS_PMF_100.i_xRemote
//     PlcTask Inputs/GVL_Devices.fb_AT1K0_GAS_PMF_100.i_xWarning <-> Channel 3/fb_AT1K0_GAS_PMF_100.i_xWarning
//   plc_kfe_gatt Instance <-> =+-CX2020/EtherCAT1/=+-EK1100_06_00/=+-ES3064_06_04
//     PlcTask Inputs/GVL_Devices.fb_AT1K0_GAS_PTM_110.i_iRawSpeed <-> AI Standard Channel 1/fb_AT1K0_GAS_PTM_110.i_iRawSpeed
//   plc_kfe_gatt Instance <-> =+-CX2020/EtherCAT1/=+-EK1100_06_00/=+-ES3064_06_06
//     PlcTask Inputs/GVL_Devices.fb_AT1K0_GAS_PTM_120.i_iCurrentMon <-> AI Standard Channel 2/fb_AT1K0_GAS_PTM_120.i_iCurrentMon
//     PlcTask Inputs/GVL_Devices.fb_AT1K0_GAS_PTM_120.i_iRawSpeed <-> AI Standard Channel 1/fb_AT1K0_GAS_PTM_120.i_iRawSpeed
//     PlcTask Inputs/GVL_Devices.fb_AT1K0_GAS_PTM_120.i_iTempMon <-> AI Standard Channel 3/fb_AT1K0_GAS_PTM_120.i_iTempMon
//   plc_kfe_gatt Instance <-> =+-CX2020/EtherCAT1/=+-EK1100_06_00/=+-ES3064_06_14
//     PlcTask Inputs/GVL_Devices.fb_AT1K0_GAS_PTM_130.i_iCurrentMon <-> AI Standard Channel 2/fb_AT1K0_GAS_PTM_130.i_iCurrentMon
//     PlcTask Inputs/GVL_Devices.fb_AT1K0_GAS_PTM_130.i_iRawSpeed <-> AI Standard Channel 1/fb_AT1K0_GAS_PTM_130.i_iRawSpeed
//     PlcTask Inputs/GVL_Devices.fb_AT1K0_GAS_PTM_130.i_iTempMon <-> AI Standard Channel 3/fb_AT1K0_GAS_PTM_130.i_iTempMon
//   plc_kfe_gatt Instance <-> =+-CX2020/EtherCAT1/=+-EK1100_06_00/=+-ES3064_06_16
//     PlcTask Inputs/GVL_Devices.fb_AT1K0_GAS_PTM_140.i_iCurrentMon <-> AI Standard Channel 2/fb_AT1K0_GAS_PTM_140.i_iCurrentMon
//     PlcTask Inputs/GVL_Devices.fb_AT1K0_GAS_PTM_140.i_iRawSpeed <-> AI Standard Channel 1/fb_AT1K0_GAS_PTM_140.i_iRawSpeed
//     PlcTask Inputs/GVL_Devices.fb_AT1K0_GAS_PTM_140.i_iTempMon <-> AI Standard Channel 3/fb_AT1K0_GAS_PTM_140.i_iTempMon
//   plc_kfe_gatt Instance <-> =+-CX2020/EtherCAT1/=+-EK1100_06_00/=+-ES4004_06_05
//     PlcTask Outputs/GVL_Devices.fb_AT1K0_GAS_PTM_110.q_iSpeedSet <-> AO Outputs Channel 1/fb_AT1K0_GAS_PTM_110.q_iSpeedSet
//     PlcTask Outputs/GVL_Devices.fb_AT1K0_GAS_PTM_120.q_iSpeedSet <-> AO Outputs Channel 3/fb_AT1K0_GAS_PTM_120.q_iSpeedSet
//   plc_kfe_gatt Instance <-> =+-CX2020/EtherCAT1/=+-EK1100_06_00/=+-ES4004_06_15
//     PlcTask Outputs/GVL_Devices.fb_AT1K0_GAS_PTM_130.q_iSpeedSet <-> AO Outputs Channel 1/fb_AT1K0_GAS_PTM_130.q_iSpeedSet
//     PlcTask Outputs/GVL_Devices.fb_AT1K0_GAS_PTM_140.q_iSpeedSet <-> AO Outputs Channel 3/fb_AT1K0_GAS_PTM_140.q_iSpeedSet
//   plc_kfe_gatt Instance <-> =+-CX2020/EtherCAT1/=+-EK1200_00_00/=+-ES2202_00_07
//     PlcTask Outputs/GVL_ILK.g_FastFaultOutput1.q_xFastFaultOut <-> Channel 1/Output
//     PlcTask Outputs/GVL_ILK.g_FastFaultOutput2.q_xFastFaultOut <-> Channel 2/Output
//   plc_kfe_gatt Instance <-> NC-Task 1 SAF/Axes/MA_1_X
//     PlcTask Inputs/Main.M1.Axis.NcToPlc <-> Outputs/ToPlc
//     PlcTask Outputs/Main.M1.Axis.PlcToNc <-> Inputs/FromPlc
//   plc_kfe_gatt Instance <-> NC-Task 1 SAF/Axes/MA_1_Y
//     PlcTask Inputs/Main.M2.Axis.NcToPlc <-> Outputs/ToPlc
//     PlcTask Outputs/Main.M2.Axis.PlcToNc <-> Inputs/FromPlc
//   plc_kfe_gatt Instance <-> NC-Task 1 SAF/Axes/MA_2_X
//     PlcTask Inputs/Main.M3.Axis.NcToPlc <-> Outputs/ToPlc
//     PlcTask Outputs/Main.M3.Axis.PlcToNc <-> Inputs/FromPlc
//   plc_kfe_gatt Instance <-> NC-Task 1 SAF/Axes/MA_2_Y
//     PlcTask Inputs/Main.M4.Axis.NcToPlc <-> Outputs/ToPlc
//     PlcTask Outputs/Main.M4.Axis.PlcToNc <-> Inputs/FromPlc
//   plc_kfe_gatt Instance <-> NC-Task 1 SAF/Axes/MA_3_X
//     PlcTask Inputs/Main.M5.Axis.NcToPlc <-> Outputs/ToPlc
//     PlcTask Outputs/Main.M5.Axis.PlcToNc <-> Inputs/FromPlc
//   plc_kfe_gatt Instance <-> NC-Task 1 SAF/Axes/MA_3_Y
//     PlcTask Inputs/Main.M6.Axis.NcToPlc <-> Outputs/ToPlc
//     PlcTask Outputs/Main.M6.Axis.PlcToNc <-> Inputs/FromPlc
//   plc_kfe_gatt Instance <-> NC-Task 1 SAF/Axes/MA_4_X
//     PlcTask Inputs/Main.M7.Axis.NcToPlc <-> Outputs/ToPlc
//     PlcTask Outputs/Main.M7.Axis.PlcToNc <-> Inputs/FromPlc
//   plc_kfe_gatt Instance <-> NC-Task 1 SAF/Axes/MA_4_Y
//     PlcTask Inputs/Main.M8.Axis.NcToPlc <-> Outputs/ToPlc
//     PlcTask Outputs/Main.M8.Axis.PlcToNc <-> Inputs/FromPlc
//   plc_kfe_gatt Instance <-> NC-Task 1 SAF/Axes/VGP_80
//     PlcTask Inputs/GVL_Devices.VGP_80.Axis.NcToPlc <-> Outputs/ToPlc
//     PlcTask Outputs/GVL_Devices.VGP_80.Axis.PlcToNc <-> Inputs/FromPlc

CONFIGURATION plc_kfe_gatt
    RESOURCE PLC ON TwinCAT3
        TASK PlcTask(INTERVAL := T#10ms, PRIORITY := 20);
        PROGRAM PRG_1_PlcTask WITH PlcTask : PRG_1_PlcTask;
    END_RESOURCE
END_CONFIGURATION

// ---- DUTs/E_HomeState.TcDUT
TYPE E_HomeState :
(
	READY,
	INIT,
	MOVING,
	MOVING2,
	CHECK,
	ERROR,
	WRITE,
	DONE
	
) UDINT;
END_TYPE

// ---- DUTs/E_MoveState.TcDUT
TYPE E_MoveState :
(
	MOVESTATE_ABORT,
	MOVESTATE_INIT,
	MOVESTATE_ENABLE,
	MOVESTATE_FORWARD,
	MOVESTATE_BACKWARDS,
	MOVESTATE_READY,
	MOVESTATE_MOVING,
	MOVESTATE_NEWTARGETPOSITION,
	MOVESTATE_NEWTARGETPOSITION2,
	MOVESTATE_ERROR,
	MOVESTATE_RESET,
	MOVESTATE_HALT,
	MOVESTATE_HOME
) UDINT;
END_TYPE

// ---- DUTs/ST_VGP.TcDUT
TYPE ST_VGP :
STRUCT

	{attribute 'pytmc' := '
    pv: POS_RDBK;
	io: i;
    '}
	// Inputs
	i_iPosition	:	REAL; //Encoder position readback (if it exists)
	{attribute 'pytmc' := '
    pv: ENC_RDBK;
	io: i;
    '}
	// Inputs
	rEnoder_Position	:	REAL; //Encoder position readback (if it exists)
	{attribute 'pytmc' := '
    pv: ERROR;
	io: i;
    '}
	// Inputs
	pv_xError	:	BOOL;
	
	{attribute 'pytmc' := '
    pv: IS_HOMED;
	io: i;
    '}
	// Inputs
	pv_xHomed	:	BOOL :=false;
	
	//Softvariables
	{attribute 'pytmc' := '
    pv: ILK_OK;
	io: i;
    '}
	xIlkOK	:	BOOL := FALSE; // Interlock Bit
	//Manually Pressing valve "Open/Close" on EDM
	{attribute 'pytmc' := '
    pv: OPN_SW;
	io: io;
    '}
	pv_xOPN_SW	: BOOL;
	
	{attribute 'pytmc' := '
    pv: GO_SW;
	io: io;
    '}
	pv_xGo_SW	: BOOL;
	
	{attribute 'pytmc' := '
    pv: HOME_SW;
	io: io;
    '}
	pv_xHome_SW	: BOOL;
	
	{attribute 'pytmc' := '
    pv: ABORT;
	io: io;
    '}
	pv_xABORT_SW	: BOOL;
	
	rUpperLimit	:	REAL:=100;	//Percentage Upper limit on valve open
	{attribute 'pytmc' := '
	pv: POS_CTRL;
	io: io; 
	'}
	rReqPosition	:	REAL; 
	// Outputs
	{attribute 'pytmc' := '
	pv: POS_DES;
	io: io;
	'}
	q_iRawPosition	:	INT; //Position control 
	{attribute 'pytmc' := '
	pv: STATE;
	type: mbbi ;
	field: ZRST CLOSE ;
	field: ONST OPEN;
	field: TWST PRESS CNTRL ;
	field: THST MANUAL CNTRL ;
	io: io;
	'}
	eValveControl	:	E_VCN := CloseValve; // Valve control state
	/// state machine state 
	{attribute 'pytmc' := '
	pv: Axis_STATE;
	io: io;
	'}
	state: E_MoveState; //Axis Move state
	ftIlk	:	F_TRIG;	

END_STRUCT
END_TYPE

// ---- GVLs/GVL_Devices.TcGVL
VAR_GLOBAL
(*AT1K0*)
/// Injector
//Valves
	{attribute 'pytmc' :=' pv: AT1K0:GAS:VCN:70 '}
	VCN_70 : FB_VCN;
	
	{attribute 'pytmc' :=' pv: AT1K0:GAS:VVC:71 '}
	VVC_71 : FB_VVC;

	{attribute 'pytmc' :=' pv: AT1K0:GAS:VVC:72 '}
	VVC_72 : FB_VVC;
	
		
	{attribute 'pytmc' :=' pv: AT1K0:GAS:VGP:80 '}
	VGP_80 : FB_VGP;

//Gauges	
	{attribute 'pytmc' :=' pv: AT1K0:GAS:GMP:70 '}
	GCM_70: FB_GCM;
	
	
	{attribute 'pytmc' :=' pv: AT1K0:GAS:GMP:80 '}
	GCM_80: FB_GCM;
	
	{attribute 'pytmc' :=' pv: AT1K0:GAS:GMP:81 '}
	GCM_81: FB_GCM;
	

	
	
	
	
	
	/////////////////////////////
	
		
	//////////////////////////////////
// MKS275 Gauges

{attribute 'pytmc' := ' pv: AT1K0:GAS:GPI:111 '}
fb_AT1K0_GAS_GPI_111 : FB_MKS275;
{attribute 'pytmc' := ' pv: AT1K0:GAS:GPI:121 '}
fb_AT1K0_GAS_GPI_121 : FB_MKS275;
{attribute 'pytmc' := ' pv: AT1K0:GAS:GPI:141 '}
fb_AT1K0_GAS_GPI_141 : FB_MKS275;

// FB_MKS317

{attribute 'pytmc' := ' pv: AT1K0:GAS:GPI:10 '}
fb_AT1K0_GAS_GPI_10 : FB_MKS317;
{attribute 'pytmc' := ' pv: AT1K0:GAS:GPI:20 '}
fb_AT1K0_GAS_GPI_20 : FB_MKS317;
{attribute 'pytmc' := ' pv: AT1K0:GAS:GPI:11 '}
fb_AT1K0_GAS_GPI_11 : FB_MKS317;
{attribute 'pytmc' := ' pv: AT1K0:GAS:GPI:30 '}
fb_AT1K0_GAS_GPI_30 : FB_MKS317;
{attribute 'pytmc' := ' pv: AT1K0:GAS:GPI:40 '}
fb_AT1K0_GAS_GPI_40 : FB_MKS317;
{attribute 'pytmc' := ' pv: AT1K0:GAS:GPI:50 '}
fb_AT1K0_GAS_GPI_50 : FB_MKS317;
{attribute 'pytmc' := ' pv: AT1K0:GAS:GPI:60 '}
fb_AT1K0_GAS_GPI_60 : FB_MKS317;
{attribute 'pytmc' := ' pv: AT1K0:GAS:GPI:51 '}
fb_AT1K0_GAS_GPI_51 : FB_MKS317;
{attribute 'pytmc' := ' pv: AT1K0:GAS:GPI:80 '}
fb_AT1K0_GAS_GPI_80 : FB_MKS317;
{attribute 'pytmc' := ' pv: AT1K0:GAS:GPI:90 '}
fb_AT1K0_GAS_GPI_90 : FB_MKS317;
{attribute 'pytmc' := ' pv: AT1K0:GAS:GPI:100 '}
fb_AT1K0_GAS_GPI_100 : FB_MKS317;
{attribute 'pytmc' := ' pv: AT1K0:GAS:GPI:110 '}
fb_AT1K0_GAS_GPI_110 : FB_MKS317;
{attribute 'pytmc' := ' pv: AT1K0:GAS:GPI:120 '}
fb_AT1K0_GAS_GPI_120 : FB_MKS317;
{attribute 'pytmc' := ' pv: AT1K0:GAS:GPI:130 '}
fb_AT1K0_GAS_GPI_130 : FB_MKS317;
{attribute 'pytmc' := ' pv: AT1K0:GAS:GPI:140 '}
fb_AT1K0_GAS_GPI_140 : FB_MKS317;

// FB_MKS422

{attribute 'pytmc' := ' pv: AT1K0:GAS:GCC:10 '}
fb_AT1K0_GAS_GCC_10 : FB_MKS422;
{attribute 'pytmc' := ' pv: AT1K0:GAS:GCC:20 '}
fb_AT1K0_GAS_GCC_20 : FB_MKS422;
{attribute 'pytmc' := ' pv: AT1K0:GAS:GCC:30 '}
fb_AT1K0_GAS_GCC_30 : FB_MKS422;
{attribute 'pytmc' := ' pv: AT1K0:GAS:GCC:40 '}
fb_AT1K0_GAS_GCC_40 : FB_MKS422;
{attribute 'pytmc' := ' pv: AT1K0:GAS:GCC:50 '}
fb_AT1K0_GAS_GCC_50 : FB_MKS422;
{attribute 'pytmc' := ' pv: AT1K0:GAS:GCC:60 '}
fb_AT1K0_GAS_GCC_60 : FB_MKS422;
{attribute 'pytmc' := ' pv: AT1K0:GAS:GCC:80 '}
fb_AT1K0_GAS_GCC_80 : FB_MKS422;
{attribute 'pytmc' := ' pv: AT1K0:GAS:GCC:90 '}
fb_AT1K0_GAS_GCC_90 : FB_MKS422;
{attribute 'pytmc' := ' pv: AT1K0:GAS:GCC:100 '}
fb_AT1K0_GAS_GCC_100 : FB_MKS422;
{attribute 'pytmc' := ' pv: AT1K0:GAS:GCC:110 '}
fb_AT1K0_GAS_GCC_110 : FB_MKS422;
{attribute 'pytmc' := ' pv: AT1K0:GAS:GCC:120 '}
fb_AT1K0_GAS_GCC_120 : FB_MKS422;
{attribute 'pytmc' := ' pv: AT1K0:GAS:GCC:130 '}
fb_AT1K0_GAS_GCC_130 : FB_MKS422;
{attribute 'pytmc' := ' pv: AT1K0:GAS:GCC:140 '}
fb_AT1K0_GAS_GCC_140 : FB_MKS422;




// FB_VRC

{attribute 'pytmc' := ' pv: AT1K0:GAS:VRC:10 '}
fb_AT1K0_GAS_VRC_10 : FB_VRC_EBD;
{attribute 'pytmc' := ' pv: AT1K0:GAS:VRC:20 '}
fb_AT1K0_GAS_VRC_20 : FB_VRC_EBD;
{attribute 'pytmc' := ' pv: AT1K0:GAS:VRC:30 '}
fb_AT1K0_GAS_VRC_30 : FB_VRC_EBD;
{attribute 'pytmc' := ' pv: AT1K0:GAS:VRC:40 '}
fb_AT1K0_GAS_VRC_40 : FB_VRC_EBD;
{attribute 'pytmc' := ' pv: AT1K0:GAS:VRC:50 '}
fb_AT1K0_GAS_VRC_50 : FB_VRC;
{attribute 'pytmc' := ' pv: AT1K0:GAS:VRC:60 '}
fb_AT1K0_GAS_VRC_60 : FB_VRC;
{attribute 'pytmc' := ' pv: AT1K0:GAS:VRC:70 '}
fb_AT1K0_GAS_VRC_70 : FB_VRC;
{attribute 'pytmc' := ' pv: AT1K0:GAS:VRC:80 '}
fb_AT1K0_GAS_VRC_80 : FB_VRC;
{attribute 'pytmc' := ' pv: AT1K0:GAS:VRC:90 '}
fb_AT1K0_GAS_VRC_90 : FB_VRC;
{attribute 'pytmc' := ' pv: AT1K0:GAS:VRC:100 '}
fb_AT1K0_GAS_VRC_100 : FB_VRC;
{attribute 'pytmc' := ' pv: AT1K0:GAS:VRC:110 '}
fb_AT1K0_GAS_VRC_110 : FB_VRC;
{attribute 'pytmc' := ' pv: AT1K0:GAS:VRC:120 '}
fb_AT1K0_GAS_VRC_120 : FB_VRC;
{attribute 'pytmc' := ' pv: AT1K0:GAS:VRC:130 '}
fb_AT1K0_GAS_VRC_130 : FB_VRC;
{attribute 'pytmc' := ' pv: AT1K0:GAS:VRC:140 '}
fb_AT1K0_GAS_VRC_140 : FB_VRC;

// PUMPS
// Turbos
// FB_PTM_Ebara_010M
{attribute 'pytmc' := ' pv: AT1K0:GAS:PTM:10 '}
fb_AT1K0_GAS_PTM_10 : FB_PTM_Ebara_010M;
{attribute 'pytmc' := ' pv: AT1K0:GAS:PTM:20 '}
fb_AT1K0_GAS_PTM_20 : FB_PTM_Ebara_010M;
{attribute 'pytmc' := ' pv: AT1K0:GAS:PTM:30 '}
fb_AT1K0_GAS_PTM_30 : FB_PTM_Ebara_010M;
{attribute 'pytmc' := ' pv: AT1K0:GAS:PTM:40 '}
fb_AT1K0_GAS_PTM_40 : FB_PTM_Ebara_010M;
{attribute 'pytmc' := ' pv: AT1K0:GAS:PTM:80 '}
fb_AT1K0_GAS_PTM_80 : FB_PTM_TwisTorr;
{attribute 'pytmc' := ' pv: AT1K0:GAS:PTM:120 '}
fb_AT1K0_GAS_PTM_120 : FB_PTM_Ebara_010M;
{attribute 'pytmc' := ' pv: AT1K0:GAS:PTM:130 '}
fb_AT1K0_GAS_PTM_130 : FB_PTM_Ebara_010M;
{attribute 'pytmc' := ' pv: AT1K0:GAS:PTM:140 '}
fb_AT1K0_GAS_PTM_140 : FB_PTM_Ebara_010M;
// FB_PTM_Ebara_011M
{attribute 'pytmc' := ' pv: AT1K0:GAS:PTM:110 '}
fb_AT1K0_GAS_PTM_110 : FB_PTM_Ebara_011M;

// Roughing
// FB_EbaraDryPump
{attribute 'pytmc' := ' pv: AT1K0:GAS:PMF:10 '}
fb_AT1K0_GAS_PMF_10 : FB_ScrollPump;
{attribute 'pytmc' := ' pv: AT1K0:GAS:PMF:60 '}
fb_AT1K0_GAS_PMF_60 : FB_ScrollPump;
{attribute 'pytmc' := ' pv: AT1K0:GAS:PMF:90 '}
fb_AT1K0_GAS_PMF_90 : FB_EbaraDryPump;
{attribute 'pytmc' := ' pv: AT1K0:GAS:PMF:100 '}
fb_AT1K0_GAS_PMF_100 : FB_EbaraDryPump;
{attribute 'pytmc' := ' pv: AT1K0:GAS:PMF:110 '}
fb_AT1K0_GAS_PMF_110 : FB_EbaraEVA;
{attribute 'pytmc' := ' pv: AT1K0:GAS:PMF:120 '}
fb_AT1K0_GAS_PMF_120 : FB_EbaraEVA;
{attribute 'pytmc' := ' pv: AT1K0:GAS:PMF:140 '}
fb_AT1K0_GAS_PMF_140 : FB_EbaraEVA;

//Roughing DC Valves
{attribute 'pytmc' := ' pv: AT1K0:GAS:VVC:110 '}
{attribute 'TcLinkTo' := 	'.q_xOPN_DO	:=	TIIB[=+-EL2212_06_25]^DOX Control Channel 1^Control^Output'}
fb_AT1K0_GAS_VVC_110 : FB_VVC;
{attribute 'pytmc' := ' pv: AT1K0:GAS:VVC:120 '}
{attribute 'TcLinkTo' := 	'.q_xOPN_DO	:=	TIIB[=+-EL2212_06_25]^DOX Control Channel 2^Control^Output'}
fb_AT1K0_GAS_VVC_120 : FB_VVC;
{attribute 'pytmc' := ' pv: AT1K0:GAS:VVC:140 '}
{attribute 'TcLinkTo' := 	'.q_xOPN_DO	:=	TIIB[=+-EL2212_06_26]^DOX Control Channel 1^Control^Output'}
fb_AT1K0_GAS_VVC_140 : FB_VVC;

END_VAR

// ---- GVLs/GVL_GATT.TcGVL
VAR_GLOBAL






END_VAR

// ---- GVLs/GVL_ILK.TcGVL
VAR_GLOBAL
	
//MPS
{attribute 'pytmc' := '
    pv: plc:lfe:gatt:FF1
    '}
    {attribute 'TcLinkTo' := '.q_xFastFaultOut:=TIIB[=+-ES2202_00_07]^Channel 1^Output'}
    g_FastFaultOutput1  :   FB_HardwareFFOutput;
	
	{attribute 'pytmc' := '
    pv: plc:lfe:gatt:FF2
    '}
    {attribute 'TcLinkTo' := '.q_xFastFaultOut:=TIIB[=+-ES2202_00_07]^Channel 2^Output'}
    g_FastFaultOutput2  :   FB_HardwareFFOutput;
	
	{attribute 'pytmc' := '
    pv: plc:kfe:FF_RESET
    '}
    xFastFaultReset :   BOOL;



	{attribute 'pytmc' := 'pv: AT1K0:GAS:VAC:OVRD_ON'}
	xSystemOverrideMode	:	BOOL; (* Global system override for the GATT*)


(* Interlock related bits, local to the PLC*)
	US_Turbo_Valves_Closed:  BOOL;
	US_Turbo_Valves_Open:  BOOL;
	DS_Turbo_Valves_Closed: BOOL;
	DS_Turbo_Valves_Open:  BOOL;
	US_Turbo_Running:  BOOL;
	DS_Turbo_Running:  BOOL;
	TwinscrewPumps_Valves_Closed: BOOL;
	US_TwinscrewPumps_Valves_Open : BOOL;
	DS_TwinscrewPumps_Valves_Open : BOOL;
	US_Aperture_Closed: BOOL;
	DS_Aperture_Closed: BOOL;
	
	xUSAperturesOpnOK : BOOL;
	xDSAperturesOpnOK : BOOL;
	
END_VAR

// ---- GVLs/GVL_MOT.TcGVL
VAR_GLOBAL
	
	//	
	

	
	
	// Array of pre defined position for every apperture on the apperture assembly array
	VAA_1_Y_POS : ARRAY [1..4]  OF LREAL;
	VAA_2_Y_POS : ARRAY [1..4]  OF LREAL;
	VAA_3_Y_POS : ARRAY [1..4]  OF LREAL;
	VAA_4_Y_POS : ARRAY [1..4]  OF LREAL;
	
	// All appertures are the same on all assemblies
	// 1 is the smallest , 4 is the biggest	
	{attribute 'pytmc' := 'pv: AT1K0:GAS:VAA:POS_DES'}
	pv_iReqApperture: INT :=1;
END_VAR

// ---- GVLs/GVL_Variables.TcGVL
VAR_GLOBAL

//xSystemOverrideMode : BOOL; (* Global system override for the prototype section*)

END_VAR

// ---- GVLs/Main.TcGVL
VAR_GLOBAL
	
	//MAA EBD
	{attribute 'pytmc' := 'pv: AT1K0:GAS_MA_X:MMS:1'}
	{attribute 'TcLinkTo' := '.bLimitForwardEnable  := TIIB[=+-ES7041_02_05]^STM Status^Status^Digital input 1;
	 						  .bLimitBackwardEnable := TIIB[=+-ES7041_02_05]^STM Status^Status^Digital input 2'}
	M1: DUT_MotionStage;
	{attribute 'pytmc' := 'pv: AT1K0:GAS_MA_Y:MMS:1'}
	{attribute 'TcLinkTo' := '.bLimitForwardEnable  := TIIB[=+-ES7041_02_06]^STM Status^Status^Digital input 2;
	 						  .bLimitBackwardEnable := TIIB[=+-ES7041_02_06]^STM Status^Status^Digital input 1;
	                          .bBrakeRelease        := TIIB[=+-ES2004_02_07]^Channel 3^Output'}
	M2: DUT_MotionStage;
	{attribute 'pytmc' := 'pv: AT1K0:GAS_MA_X:MMS:2'}
	{attribute 'TcLinkTo' := '.bLimitForwardEnable  := TIIB[=+-ES7041_02_09]^STM Status^Status^Digital input 1;
	 						  .bLimitBackwardEnable := TIIB[=+-ES7041_02_09]^STM Status^Status^Digital input 2'}
	M3: DUT_MotionStage;
	{attribute 'pytmc' := 'pv: AT1K0:GAS_MA_Y:MMS:2'}
	{attribute 'TcLinkTo' := '.bLimitForwardEnable  := TIIB[=+-ES7041_02_10]^STM Status^Status^Digital input 2;
	 						  .bLimitBackwardEnable := TIIB[=+-ES7041_02_10]^STM Status^Status^Digital input 1;
	                          .bBrakeRelease        := TIIB[=+-ES2004_02_07]^Channel 4^Output'}
	M4: DUT_MotionStage;
	//MAA FEE
	
	{attribute 'pytmc' := 'pv: AT1K0:GAS_MA_X:MMS:3'}
	{attribute 'TcLinkTo' := '.bLimitForwardEnable  := TIIB[=+-EL7041_04_07]^STM Status^Status^Digital input 2;
	 						  .bLimitBackwardEnable := TIIB[=+-EL7041_04_07]^STM Status^Status^Digital input 1;
	                          .bBrakeRelease        := TIIB[=+-ES2004_04_09]^Channel 1^Output'}
	M5: DUT_MotionStage;
	{attribute 'pytmc' := 'pv: AT1K0:GAS_MA_Y:MMS:3'}
	{attribute 'TcLinkTo' := '.bLimitForwardEnable  := TIIB[=+-EL7041_04_08]^STM Status^Status^Digital input 2;
	 						  .bLimitBackwardEnable := TIIB[=+-EL7041_04_08]^STM Status^Status^Digital input 1;
	                          .bBrakeRelease        := TIIB[=+-ES2004_04_09]^Channel 2^Output'}
	M6: DUT_MotionStage;
	{attribute 'pytmc' := 'pv: AT1K0:GAS_MA_X:MMS:4'}
	{attribute 'TcLinkTo' := '.bLimitForwardEnable  := TIIB[=+-EL7041_04_10]^STM Status^Status^Digital input 2;
	 						  .bLimitBackwardEnable := TIIB[=+-EL7041_04_10]^STM Status^Status^Digital input 1;
	                          .bBrakeRelease        := TIIB[=+-ES2004_04_09]^Channel 3^Output'}
	M7: DUT_MotionStage;
	{attribute 'pytmc' := 'pv: AT1K0:GAS_MA_Y:MMS:4'}
	{attribute 'TcLinkTo' := '.bLimitForwardEnable  := TIIB[=+-EL7041_04_11]^STM Status^Status^Digital input 2;
	 						  .bLimitBackwardEnable := TIIB[=+-EL7041_04_11]^STM Status^Status^Digital input 1;
	                          .bBrakeRelease        := TIIB[=+-ES2004_04_09]^Channel 4^Output'}
	M8: DUT_MotionStage;
	
END_VAR

// ---- POUs/PRG_1_PlcTask.TcPOU
PROGRAM PRG_1_PlcTask
VAR
	
	
END_VAR

(*Ethercat Diagnostics*)
//DIAGNOSTICS();

PRG_Motors_Test();

// Functionblock for PTP motion between different appertures
//PRG_Motion();

// Vacuum and differential pumping
PRG_GATT();
// Injector
PRG_INJ();

//PRG_VGP();

END_PROGRAM

// ---- POUs/PRG_Motors_Test.TcPOU
PROGRAM PRG_Motors_Test
VAR

	Y1_Power: MC_Power;
	Y2_Power: MC_Power;
	Y3_Power: MC_Power;
	Y4_Power: MC_Power;
	X1_Power: MC_Power;
	X2_Power: MC_Power;
	X3_Power: MC_Power;
	X4_Power: MC_Power;
	
	
	Y1_ENC AT%I* :INT;
	Y2_ENC AT%I* :INT;
	Y3_ENC AT%I* :INT;
	Y4_ENC AT%I* :INT;
	X1_ENC AT%I* :INT;
	X2_ENC AT%I* :INT;
	X3_ENC AT%I* :INT;
	X4_ENC AT%I* :INT;
	
END_VAR

X1_Power(//reverse motor direction?
	Axis:=  M1.Axis, 
	Enable:= M1.bBrakeRelease, 
	Enable_Positive:= M1.bLimitForwardEnable, // fix
	Enable_Negative:= M1.bLimitBackwardEnable,  // fix -- verify
	Override:= , 
	BufferMode:= , 
	Options:= , 
	Status=> , 
	Busy=> , 
	Active=> , 
	Error=> , 
	ErrorID=> );

Y1_Power(
	Axis:=  M2.Axis, 
	Enable:= M2.bBrakeRelease, 
	Enable_Positive:= M2.bLimitForwardEnable, 
	Enable_Negative:= M2.bLimitBackwardEnable, 
	Override:= , 
	BufferMode:= , 
	Options:= , 
	Status=> , 
	Busy=> , 
	Active=> , 
	Error=> , 
	ErrorID=> );
	
	
	
X2_Power(
	Axis:=  M3.Axis, 
	Enable:= M3.bBrakeRelease, 
	Enable_Positive:= M3.bLimitForwardEnable, // fix
	Enable_Negative:= M3.bLimitBackwardEnable,  // fix -- verify
	Override:= , 
	BufferMode:= , 
	Options:= , 
	Status=> , 
	Busy=> , 
	Active=> , 
	Error=> , 
	ErrorID=> );	
	
Y2_Power(
	Axis:=  M4.Axis, 
	Enable:= M4.bBrakeRelease, 
	Enable_Positive:= M4.bLimitForwardEnable, 
	Enable_Negative:= M4.bLimitBackwardEnable, 
	Override:= , 
	BufferMode:= , 
	Options:= , 
	Status=> , 
	Busy=> , 
	Active=> , 
	Error=> , 
	ErrorID=> );
	
X3_Power(
	Axis:=  M5.Axis, 
	Enable:= M5.bBrakeRelease, 
	Enable_Positive:= M5.bLimitForwardEnable, 
	Enable_Negative:= M5.bLimitBackwardEnable,  
	Override:= , 
	BufferMode:= , 
	Options:= , 
	Status=> , 
	Busy=> , 
	Active=> , 
	Error=> , 
	ErrorID=> );
Y3_Power(
	Axis:=  M6.Axis, 
	Enable:= M6.bBrakeRelease, 
	Enable_Positive:= M6.bLimitForwardEnable, 
	Enable_Negative:= M6.bLimitBackwardEnable, 
	Override:= , 
	BufferMode:= , 
	Options:= , 
	Status=> , 
	Busy=> , 
	Active=> , 
	Error=> , 
	ErrorID=> );
	
	
X4_Power(
	Axis:=  M7.Axis, 
	Enable:= M7.bBrakeRelease, 
	Enable_Positive:= M7.bLimitForwardEnable, 
	Enable_Negative:= M7.bLimitBackwardEnable,  
	Override:= , 
	BufferMode:= , 
	Options:= , 
	Status=> , 
	Busy=> , 
	Active=> , 
	Error=> , 
	ErrorID=> );
Y4_Power(
	Axis:=  M8.Axis, 
	Enable:= M8.bBrakeRelease, 
	Enable_Positive:= M8.bLimitForwardEnable, 
	Enable_Negative:= M8.bLimitBackwardEnable, 
	Override:= , 
	BufferMode:= , 
	Options:= , 
	Status=> , 
	Busy=> , 
	Active=> , 
	Error=> , 
	ErrorID=> );

END_PROGRAM

// ---- POUs/PRG_GATT.TcPOU
PROGRAM PRG_GATT
VAR
END_VAR



// GAUGES
// MKS275 Gauges
fb_AT1K0_GAS_GPI_111(PG=>);
fb_AT1K0_GAS_GPI_121(PG=>);
fb_AT1K0_GAS_GPI_141(PG=>);
// FB_MKS317
fb_AT1K0_GAS_GPI_10(PG=>);
fb_AT1K0_GAS_GPI_20(PG=>);
fb_AT1K0_GAS_GPI_11(PG=>);
fb_AT1K0_GAS_GPI_30(PG=>);
fb_AT1K0_GAS_GPI_40(PG=>);
fb_AT1K0_GAS_GPI_50(PG=>);
fb_AT1K0_GAS_GPI_51(PG=>);
fb_AT1K0_GAS_GPI_60(PG=>);
fb_AT1K0_GAS_GPI_80(PG=>);
fb_AT1K0_GAS_GPI_90(PG=>);
fb_AT1K0_GAS_GPI_100(PG=>);
fb_AT1K0_GAS_GPI_110(PG=>);
fb_AT1K0_GAS_GPI_120(PG=>);
fb_AT1K0_GAS_GPI_130(PG=>);
fb_AT1K0_GAS_GPI_140(PG=>);

// FB_MKS422

fb_AT1K0_GAS_GCC_10(PG := fb_AT1K0_GAS_GPI_10.PG);
fb_AT1K0_GAS_GCC_20(PG := fb_AT1K0_GAS_GPI_20.PG);
fb_AT1K0_GAS_GCC_30(PG := fb_AT1K0_GAS_GPI_30.PG);
fb_AT1K0_GAS_GCC_40(PG := fb_AT1K0_GAS_GPI_40.PG);
fb_AT1K0_GAS_GCC_50(PG := fb_AT1K0_GAS_GPI_50.PG);
fb_AT1K0_GAS_GCC_60(PG := fb_AT1K0_GAS_GPI_60.PG);
fb_AT1K0_GAS_GCC_80(PG := fb_AT1K0_GAS_GPI_80.PG);
fb_AT1K0_GAS_GCC_90(PG := fb_AT1K0_GAS_GPI_90.PG);
fb_AT1K0_GAS_GCC_100(PG := fb_AT1K0_GAS_GPI_100.PG);
fb_AT1K0_GAS_GCC_110(PG := fb_AT1K0_GAS_GPI_110.PG);
fb_AT1K0_GAS_GCC_120(PG := fb_AT1K0_GAS_GPI_120.PG);
fb_AT1K0_GAS_GCC_130(PG := fb_AT1K0_GAS_GPI_130.PG);
fb_AT1K0_GAS_GCC_140(PG := fb_AT1K0_GAS_GPI_140.PG);


//VALVES
// Pump Isolation Valves
// FB_VRC
fb_AT1K0_GAS_VRC_10(i_xExtILK_OK := F_TurboGateValve_ILK(fb_AT1K0_GAS_PTM_10.iq_stPtm,fb_AT1K0_GAS_GPI_10.PG), i_xOverrideMode := xSystemOverrideMode);
fb_AT1K0_GAS_VRC_20(i_xExtILK_OK := F_TurboGateValve_ILK(fb_AT1K0_GAS_PTM_20.iq_stPtm,fb_AT1K0_GAS_GPI_20.PG) , i_xOverrideMode := xSystemOverrideMode);
fb_AT1K0_GAS_VRC_30(i_xExtILK_OK := F_TurboGateValve_ILK(fb_AT1K0_GAS_PTM_30.iq_stPtm,fb_AT1K0_GAS_GPI_30.PG), i_xOverrideMode := xSystemOverrideMode);
fb_AT1K0_GAS_VRC_40(i_xExtILK_OK := F_TurboGateValve_ILK(fb_AT1K0_GAS_PTM_40.iq_stPtm,fb_AT1K0_GAS_GPI_40.PG), i_xOverrideMode := xSystemOverrideMode);
fb_AT1K0_GAS_VRC_50(i_xExtILK_OK := fb_AT1K0_GAS_PMF_60.iq_stPFO.q_xRunDo , i_xOverrideMode := xSystemOverrideMode);
fb_AT1K0_GAS_VRC_60(i_xExtILK_OK := fb_AT1K0_GAS_PMF_60.iq_stPFO.q_xRunDo, i_xOverrideMode := xSystemOverrideMode);
fb_AT1K0_GAS_VRC_70(i_xExtILK_OK := fb_AT1K0_GAS_PMF_100.stPump.i_xMPStatus, i_xOverrideMode := xSystemOverrideMode);
fb_AT1K0_GAS_VRC_90(i_xExtILK_OK := fb_AT1K0_GAS_PMF_100.stPump.i_xMPStatus, i_xOverrideMode := xSystemOverrideMode);
fb_AT1K0_GAS_VRC_100(i_xExtILK_OK := fb_AT1K0_GAS_PMF_100.stPump.i_xMPStatus, i_xOverrideMode := xSystemOverrideMode);
fb_AT1K0_GAS_VRC_110(i_xExtILK_OK := F_TurboGateValve_ILK(fb_AT1K0_GAS_PTM_110.iq_stPtm,fb_AT1K0_GAS_GPI_110.PG), i_xOverrideMode := xSystemOverrideMode);
fb_AT1K0_GAS_VRC_120(i_xExtILK_OK := F_TurboGateValve_ILK(fb_AT1K0_GAS_PTM_120.iq_stPtm,fb_AT1K0_GAS_GPI_120.PG), i_xOverrideMode := xSystemOverrideMode);
fb_AT1K0_GAS_VRC_130(i_xExtILK_OK := F_TurboGateValve_ILK(fb_AT1K0_GAS_PTM_130.iq_stPtm,fb_AT1K0_GAS_GPI_130.PG), i_xOverrideMode := xSystemOverrideMode);
fb_AT1K0_GAS_VRC_140(i_xExtILK_OK :=F_TurboGateValve_ILK(fb_AT1K0_GAS_PTM_140.iq_stPtm,fb_AT1K0_GAS_GPI_140.PG) , i_xOverrideMode := xSystemOverrideMode);
//N2 valve
//INL VCN, VGP and VRC_70 are closed.
fb_AT1K0_GAS_VRC_80.i_xExtILK_OK := fb_AT1K0_GAS_VRC_90.iq_stValve.i_xClsLS AND VCN_70.iq_stVCN.rReqPosition <0.4; //AND VGP is closed;
fb_AT1K0_GAS_VRC_80( i_xOverrideMode := xSystemOverrideMode);


// Turbo Pumps
// FB_PTM_Ebara_010M
fb_AT1K0_GAS_PTM_10(i_xExtILKOk := F_TurboExtILKLogic_2(fb_AT1K0_GAS_PTM_10.iq_stPtm, fb_AT1K0_GAS_GPI_11.PG, fb_AT1K0_GAS_GPI_10.PG,fb_AT1K0_GAS_PMF_10.iq_stPFO));
fb_AT1K0_GAS_PTM_20(i_xExtILKOk := F_TurboExtILKLogic_2(fb_AT1K0_GAS_PTM_20.iq_stPtm, fb_AT1K0_GAS_GPI_11.PG, fb_AT1K0_GAS_GPI_20.PG,fb_AT1K0_GAS_PMF_10.iq_stPFO));
fb_AT1K0_GAS_PTM_30(i_xExtILKOk := F_TurboExtILKLogic_2(fb_AT1K0_GAS_PTM_30.iq_stPtm, fb_AT1K0_GAS_GPI_11.PG, fb_AT1K0_GAS_GPI_30.PG,fb_AT1K0_GAS_PMF_10.iq_stPFO));
fb_AT1K0_GAS_PTM_40(i_xExtILKOk := F_TurboExtILKLogic_2(fb_AT1K0_GAS_PTM_40.iq_stPtm, fb_AT1K0_GAS_GPI_11.PG, fb_AT1K0_GAS_GPI_40.PG,fb_AT1K0_GAS_PMF_10.iq_stPFO));
fb_AT1K0_GAS_PTM_110(i_xExtILKOk := F_TurboExtILKLogic_2(fb_AT1K0_GAS_PTM_110.iq_stPtm, fb_AT1K0_GAS_GPI_111.PG,fb_AT1K0_GAS_GPI_110.PG,fb_AT1K0_GAS_PMF_110.stPump));
fb_AT1K0_GAS_PTM_120(i_xExtILKOk := F_TurboExtILKLogic_2(fb_AT1K0_GAS_PTM_120.iq_stPtm, fb_AT1K0_GAS_GPI_121.PG, fb_AT1K0_GAS_GPI_120.PG,fb_AT1K0_GAS_PMF_120.stPump));
fb_AT1K0_GAS_PTM_130(i_xExtILKOk := F_TurboExtILKLogic_2(fb_AT1K0_GAS_PTM_130.iq_stPtm, fb_AT1K0_GAS_GPI_121.PG,fb_AT1K0_GAS_GPI_130.PG,fb_AT1K0_GAS_PMF_120.stPump)); 
fb_AT1K0_GAS_PTM_140(i_xExtILKOk := F_TurboExtILKLogic_2(fb_AT1K0_GAS_PTM_140.iq_stPtm, fb_AT1K0_GAS_GPI_141.PG,fb_AT1K0_GAS_GPI_140.PG,fb_AT1K0_GAS_PMF_140.stPump));



